gfCNCPoint5[15643] = {X -1.0364, Y 9.9250, Z -7.1667, A 0.000, B 0.000, C 0.000 }
gfCNCPoint5[15644] = {X -0.1703, Y 9.5539, Z -7.1667, A 0.000, B 0.000, C 0.000 }
gfCNCPoint5[15645] = {X 0.7570, Y 9.3871, Z -7.1667, A 0.000, B 0.000, C 0.000 }
gfCNCPoint5[15646] = {X 1.6981, Y 9.4333, Z -7.1667, A 0.000, B 0.000, C 0.000 }
gfCNCPoint5[15647] = {X 2.6047, Y 9.6901, Z -7.1667, A 0.000, B 0.000, C 0.000 }
gfCNCPoint5[15648] = {X 3.5530, Y 9.2659, Z -7.1667, A 0.000, B 0.000, C 0.000 }
gfCNCPoint5[15649] = {X 5.6159, Y 8.4887, Z -7.1667, A 0.000, B 0.000, C 0.000 }
gfCNCPoint5[15650] = {X 7.7422, Y 7.9071, Z -7.1667, A 0.000, B 0.000, C 0.000 }
gfCNCPoint5[15651] = {X 9.9135, Y 7.5260, Z -7.1667, A 0.000, B 0.000, C 0.000 }
gfCNCPoint5[15652] = {X 12.1108, Y 7.3488, Z -7.1667, A 0.000, B 0.000, C 0.000 }
gfCNCPoint5[15653] = {X 14.3150, Y 7.3770, Z -7.1667, A 0.000, B 0.000, C 0.000 }
gfCNCPoint5[15654] = {X 16.5070, Y 7.6105, Z -7.1667, A 0.000, B 0.000, C 0.000 }
gfCNCPoint5[15655] = {X 18.2265, Y 7.9626, Z -7.1667, A 0.000, B 0.000, C 0.000 }
gfCNCPoint5[15656] = {X 19.9014, Y 8.4872, Z -7.1667, A 0.000, B 0.000, C 0.000 }
gfCNCPoint5[15657] = {X 21.5145, Y 9.1790, Z -7.1667, A 0.000, B 0.000, C 0.000 }
gfCNCPoint5[15658] = {X 23.0491, Y 10.0308, Z -7.1667, A 0.000, B 0.000, C 0.000 }
gfCNCPoint5[15659] = {X 24.4894, Y 11.0338, Z -7.1667, A 0.000, B 0.000, C 0.000 }
gfCNCPoint5[15660] = {X 25.5613, Y 11.9712, Z -7.1667, A 0.000, B 0.000, C 0.000 }
gfCNCPoint5[15661] = {X 26.5229, Y 13.0215, Z -7.1667, A 0.000, B 0.000, C 0.000 }
gfCNCPoint5[15662] = {X 27.3624, Y 14.1717, Z -7.1667, A 0.000, B 0.000, C 0.000 }
gfCNCPoint5[15663] = {X 28.0693, Y 15.4079, Z -7.1667, A 0.000, B 0.000, C 0.000 }
gfCNCPoint5[15664] = {X 28.6351, Y 16.7147, Z -7.1667, A 0.000, B 0.000, C 0.000 }
gfCNCPoint5[15665] = {X 29.1044, Y 18.3529, Z -7.1667, A 0.000, B 0.000, C 0.000 }
gfCNCPoint5[15666] = {X 29.3828, Y 20.0341, Z -7.1667, A 0.000, B 0.000, C 0.000 }
gfCNCPoint5[15667] = {X 29.4668, Y 21.7361, Z -7.1667, A 0.000, B 0.000, C 0.000 }
gfCNCPoint5[15668] = {X 29.3551, Y 23.4365, Z -7.1667, A 0.000, B 0.000, C 0.000 }
gfCNCPoint5[15669] = {X 29.0493, Y 25.1129, Z -7.1667, A 0.000, B 0.000, C 0.000 }
gfCNCPoint5[15670] = {X 28.6229, Y 26.5132, Z -7.1667, A 0.000, B 0.000, C 0.000 }
gfCNCPoint5[15671] = {X 28.0227, Y 27.8482, Z -7.1667, A 0.000, B 0.000, C 0.000 }
gfCNCPoint5[15672] = {X 27.2582, Y 29.0964, Z -7.1667, A 0.000, B 0.000, C 0.000 }
gfCNCPoint5[15673] = {X 26.3417, Y 30.2377, Z -7.1667, A 0.000, B 0.000, C 0.000 }
gfCNCPoint5[15674] = {X 25.2881, Y 31.2538, Z -7.1667, A 0.000, B 0.000, C 0.000 }
gfCNCPoint5[15675] = {X 25.1139, Y 31.3987, Z -7.1667, A 0.000, B 0.000, C 0.000 }
gfCNCPoint5[15676] = {X 24.9369, Y 31.5402, Z -7.1667, A 0.000, B 0.000, C 0.000 }
gfCNCPoint5[15677] = {X 25.8030, Y 31.8442, Z -7.1667, A 0.000, B 0.000, C 0.000 }
gfCNCPoint5[15678] = {X 26.5813, Y 32.3308, Z -7.1667, A 0.000, B 0.000, C 0.000 }
gfCNCPoint5[15679] = {X 27.2339, Y 32.9762, Z -7.1667, A 0.000, B 0.000, C 0.000 }
gfCNCPoint5[15680] = {X 27.7292, Y 33.7491, Z -7.1667, A 0.000, B 0.000, C 0.000 }
gfCNCPoint5[15681] = {X 30.7660, Y 40.0227, Z -7.1667, A 0.000, B 0.000, C 0.000 }
gfCNCPoint5[15682] = {X 31.0747, Y 40.8982, Z -7.1667, A 0.000, B 0.000, C 0.000 }
gfCNCPoint5[15683] = {X 31.1815, Y 41.8203, Z -7.1667, A 0.000, B 0.000, C 0.000 }
gfCNCPoint5[15684] = {X 31.0813, Y 42.7431, Z -7.1667, A 0.000, B 0.000, C 0.000 }
gfCNCPoint5[15685] = {X 30.7789, Y 43.6208, Z -7.1667, A 0.000, B 0.000, C 0.000 }
gfCNCPoint5[15686] = {X 30.2893, Y 44.4095, Z -7.1667, A 0.000, B 0.000, C 0.000 }
gfCNCPoint5[15687] = {X 29.6371, Y 45.0700, Z -7.1667, A 0.000, B 0.000, C 0.000 }
gfCNCPoint5[15688] = {X 29.1011, Y 45.5034, Z -7.1667, A 0.000, B 0.000, C 0.000 }
gfCNCPoint5[15689] = {X 28.4112, Y 45.9565, Z -7.1667, A 0.000, B 0.000, C 0.000 }
gfCNCPoint5[15690] = {X 27.6455, Y 46.2648, Z -7.1667, A 0.000, B 0.000, C 0.000 }
gfCNCPoint5[15691] = {X 26.8342, Y 46.4162, Z -7.1667, A 0.000, B 0.000, C 0.000 }
gfCNCPoint5[15692] = {X 26.0089, Y 46.4050, Z -7.1667, A 0.000, B 0.000, C 0.000 }
gfCNCPoint5[15693] = {X 25.2019, Y 46.2314, Z -7.1667, A 0.000, B 0.000, C 0.000 }
gfCNCPoint5[15694] = {X 23.3925, Y 47.1909, Z -7.1667, A 0.000, B 0.000, C 0.000 }
gfCNCPoint5[15695] = {X 21.5199, Y 48.0206, Z -7.1667, A 0.000, B 0.000, C 0.000 }
gfCNCPoint5[15696] = {X 19.5936, Y 48.7163, Z -7.1667, A 0.000, B 0.000, C 0.000 }
gfCNCPoint5[15697] = {X 17.6674, Y 49.2600, Z -7.1667, A 0.000, B 0.000, C 0.000 }
gfCNCPoint5[15698] = {X 15.7006, Y 49.6311, Z -7.1667, A 0.000, B 0.000, C 0.000 }
gfCNCPoint5[15699] = {X 13.7087, Y 49.8267, Z -7.1667, A 0.000, B 0.000, C 0.000 }
gfCNCPoint5[15700] = {X 11.7074, Y 49.8453, Z -7.1667, A 0.000, B 0.000, C 0.000 }
gfCNCPoint5[15701] = {X 9.7122, Y 49.6868, Z -7.1667, A 0.000, B 0.000, C 0.000 }
gfCNCPoint5[15702] = {X 7.7389, Y 49.3523, Z -7.1667, A 0.000, B 0.000, C 0.000 }
gfCNCPoint5[15703] = {X 5.8554, Y 48.8363, Z -7.1667, A 0.000, B 0.000, C 0.000 }
gfCNCPoint5[15704] = {X 4.0458, Y 48.1022, Z -7.1667, A 0.000, B 0.000, C 0.000 }
gfCNCPoint5[15705] = {X 2.3352, Y 47.1601, Z -7.1667, A 0.000, B 0.000, C 0.000 }
gfCNCPoint5[15706] = {X 0.7475, Y 46.0231, Z -7.1667, A 0.000, B 0.000, C 0.000 }
gfCNCPoint5[15707] = {X -0.3710, Y 45.0177, Z -7.1667, A 0.000, B 0.000, C 0.000 }
gfCNCPoint5[15708] = {X -1.3644, Y 43.8885, Z -7.1667, A 0.000, B 0.000, C 0.000 }
gfCNCPoint5[15709] = {X -2.2192, Y 42.6512, Z -7.1667, A 0.000, B 0.000, C 0.000 }
gfCNCPoint5[15710] = {X -2.9237, Y 41.3225, Z -7.1667, A 0.000, B 0.000, C 0.000 }
gfCNCPoint5[15711] = {X -3.4683, Y 39.9206, Z -7.1667, A 0.000, B 0.000, C 0.000 }
gfCNCPoint5[15712] = {X -3.5888, Y 39.5251, Z -7.1667, A 0.000, B 0.000, C 0.000 }
gfCNCPoint5[15713] = {X -3.6967, Y 39.1259, Z -7.1667, A 0.000, B 0.000, C 0.000 }
gfCNCPoint5[15714] = {X -4.6774, Y 35.2480, Z -7.1667, A 0.000, B 0.000, C 0.000 }
gfCNCPoint5[15715] = {X -8.0069, Y 35.2272, Z -7.1667, A 0.000, B 0.000, C 0.000 }
gfCNCPoint5[15716] = {X -8.0069, Y 35.2272, Z -4.1667, A 0.000, B 0.000, C 0.000 }
gfCNCPoint5[15717] = {X -8.0069, Y 35.2272, Z 11.0000, A 0.000, B 0.000, C 0.000 }
gfCNCPoint5[15718] = {X -7.9995, Y 34.8056, Z 11.0000, A 0.000, B 0.000, C 0.000 }
gfCNCPoint5[15719] = {X -7.9995, Y 34.8056, Z -4.1667, A 0.000, B 0.000, C 0.000 }
gfCNCPoint5[15720] = {X -7.9995, Y 34.8056, Z -7.1667, A 0.000, B 0.000, C 0.000 }
gfCNCPoint5[15721] = {X -4.8517, Y 34.8970, Z -7.1667, A 0.000, B 0.000, C 0.000 }
gfCNCPoint5[15722] = {X -3.6967, Y 31.0674, Z -7.1667, A 0.000, B 0.000, C 0.000 }
gfCNCPoint5[15723] = {X -3.6591, Y 30.9448, Z -7.1667, A 0.000, B 0.000, C 0.000 }
gfCNCPoint5[15724] = {X -3.6205, Y 30.8225, Z -7.1667, A 0.000, B 0.000, C 0.000 }
gfCNCPoint5[15725] = {X -3.4458, Y 30.3101, Z -7.1667, A 0.000, B 0.000, C 0.000 }
gfCNCPoint5[15726] = {X -3.2526, Y 29.8045, Z -7.1667, A 0.000, B 0.000, C 0.000 }
gfCNCPoint5[15727] = {X -2.6179, Y 28.4651, Z -7.1667, A 0.000, B 0.000, C 0.000 }
gfCNCPoint5[15728] = {X -1.8063, Y 27.2249, Z -7.1667, A 0.000, B 0.000, C 0.000 }
gfCNCPoint5[15729] = {X -0.8329, Y 26.1072, Z -7.1667, A 0.000, B 0.000, C 0.000 }
gfCNCPoint5[15730] = {X 0.2840, Y 25.1328, Z -7.1667, A 0.000, B 0.000, C 0.000 }
gfCNCPoint5[15731] = {X 1.5235, Y 24.3201, Z -7.1667, A 0.000, B 0.000, C 0.000 }
gfCNCPoint5[15732] = {X 0.7354, Y 23.9293, Z -7.1667, A 0.000, B 0.000, C 0.000 }
gfCNCPoint5[15733] = {X 0.0428, Y 23.3868, Z -7.1667, A 0.000, B 0.000, C 0.000 }
gfCNCPoint5[15734] = {X -0.5255, Y 22.7154, Z -7.1667, A 0.000, B 0.000, C 0.000 }
gfCNCPoint5[15735] = {X -0.9460, Y 21.9427, Z -7.1667, A 0.000, B 0.000, C 0.000 }
gfCNCPoint5[15736] = {X -3.6217, Y 15.3839, Z -7.1667, A 0.000, B 0.000, C 0.000 }
gfCNCPoint5[15737] = {X -3.6606, Y 15.2745, Z -7.1667, A 0.000, B 0.000, C 0.000 }
gfCNCPoint5[15738] = {X -3.6967, Y 15.1642, Z -7.1667, A 0.000, B 0.000, C 0.000 }
gfCNCPoint5[15739] = {X -4.8865, Y 11.3452, Z -7.1667, A 0.000, B 0.000, C 0.000 }
gfCNCPoint5[15740] = {X -7.6967, Y 11.3452, Z -7.1667, A 0.000, B 0.000, C 0.000 }
gfCNCPoint5[15741] = {X -7.6967, Y 11.3452, Z -4.1667, A 0.000, B 0.000, C 0.000 }
gfCNCPoint5[15742] = {X -7.6967, Y 11.3452, Z 11.0000, A 0.000, B 0.000, C 0.000 }
gfCNCPoint5[15743] = {X -8.0065, Y 35.1744, Z 11.0000, A 0.000, B 0.000, C 0.000 }
gfCNCPoint5[15744] = {X -8.0065, Y 35.1744, Z -4.1667, A 0.000, B 0.000, C 0.000 }
gfCNCPoint5[15745] = {X -8.0065, Y 35.1744, Z -7.1667, A 0.000, B 0.000, C 0.000 }
gfCNCPoint5[15746] = {X -4.7803, Y 35.2037, Z -7.1667, A 0.000, B 0.000, C 0.000 }
gfCNCPoint5[15747] = {X -3.6967, Y 31.3533, Z -7.1667, A 0.000, B 0.000, C 0.000 }
gfCNCPoint5[15748] = {X -3.6228, Y 31.0994, Z -7.1667, A 0.000, B 0.000, C 0.000 }
gfCNCPoint5[15749] = {X -3.5443, Y 30.8469, Z -7.1667, A 0.000, B 0.000, C 0.000 }
gfCNCPoint5[15750] = {X -3.3705, Y 30.3371, Z -7.1667, A 0.000, B 0.000, C 0.000 }
gfCNCPoint5[15751] = {X -3.1782, Y 29.8341, Z -7.1667, A 0.000, B 0.000, C 0.000 }
gfCNCPoint5[15752] = {X -2.5643, Y 28.5332, Z -7.1667, A 0.000, B 0.000, C 0.000 }
gfCNCPoint5[15753] = {X -1.7821, Y 27.3259, Z -7.1667, A 0.000, B 0.000, C 0.000 }
gfCNCPoint5[15754] = {X -0.8458, Y 26.2339, Z -7.1667, A 0.000, B 0.000, C 0.000 }
gfCNCPoint5[15755] = {X 0.2280, Y 25.2767, Z -7.1667, A 0.000, B 0.000, C 0.000 }
gfCNCPoint5[15756] = {X 1.4199, Y 24.4715, Z -7.1667, A 0.000, B 0.000, C 0.000 }
gfCNCPoint5[15757] = {X 1.5687, Y 24.3865, Z -7.1667, A 0.000, B 0.000, C 0.000 }
gfCNCPoint5[15758] = {X 1.7187, Y 24.3039, Z -7.1667, A 0.000, B 0.000, C 0.000 }
gfCNCPoint5[15759] = {X 0.8916, Y 23.9307, Z -7.1667, A 0.000, B 0.000, C 0.000 }
gfCNCPoint5[15760] = {X 0.1628, Y 23.3900, Z -7.1667, A 0.000, B 0.000, C 0.000 }
gfCNCPoint5[15761] = {X -0.4342, Y 22.7066, Z -7.1667, A 0.000, B 0.000, C 0.000 }
gfCNCPoint5[15762] = {X -0.8722, Y 21.9118, Z -7.1667, A 0.000, B 0.000, C 0.000 }
gfCNCPoint5[15763] = {X -3.5467, Y 15.3560, Z -7.1667, A 0.000, B 0.000, C 0.000 }
gfCNCPoint5[15764] = {X -3.6292, Y 15.1114, Z -7.1667, A 0.000, B 0.000, C 0.000 }
gfCNCPoint5[15765] = {X -3.6967, Y 14.8622, Z -7.1667, A 0.000, B 0.000, C 0.000 }
gfCNCPoint5[15766] = {X -4.6241, Y 10.9713, Z -7.1667, A 0.000, B 0.000, C 0.000 }
gfCNCPoint5[15767] = {X -7.6967, Y 10.9713, Z -7.1667, A 0.000, B 0.000, C 0.000 }
gfCNCPoint5[15768] = {X -7.6967, Y 10.9713, Z -4.1667, A 0.000, B 0.000, C 0.000 }
gfCNCPoint5[15769] = {X -7.6967, Y 10.9713, Z 11.0000, A 0.000, B 0.000, C 0.000 }
gfCNCPoint5[15770] = {X -8.0058, Y 35.5721, Z 11.0000, A 0.000, B 0.000, C 0.000 }
gfCNCPoint5[15771] = {X -8.0058, Y 35.5721, Z -4.1667, A 0.000, B 0.000, C 0.000 }
gfCNCPoint5[15772] = {X -8.0058, Y 35.5721, Z -7.1667, A 0.000, B 0.000, C 0.000 }
gfCNCPoint5[15773] = {X -4.7025, Y 35.5310, Z -7.1667, A 0.000, B 0.000, C 0.000 }
gfCNCPoint5[15774] = {X -3.6967, Y 31.6595, Z -7.1667, A 0.000, B 0.000, C 0.000 }
gfCNCPoint5[15775] = {X -3.5879, Y 31.2638, Z -7.1667, A 0.000, B 0.000, C 0.000 }
gfCNCPoint5[15776] = {X -3.4681, Y 30.8713, Z -7.1667, A 0.000, B 0.000, C 0.000 }
gfCNCPoint5[15777] = {X -3.2952, Y 30.3642, Z -7.1667, A 0.000, B 0.000, C 0.000 }
gfCNCPoint5[15778] = {X -3.1039, Y 29.8636, Z -7.1667, A 0.000, B 0.000, C 0.000 }
gfCNCPoint5[15779] = {X -2.4945, Y 28.5724, Z -7.1667, A 0.000, B 0.000, C 0.000 }
gfCNCPoint5[15780] = {X -1.7182, Y 27.3740, Z -7.1667, A 0.000, B 0.000, C 0.000 }
gfCNCPoint5[15781] = {X -0.7888, Y 26.2901, Z -7.1667, A 0.000, B 0.000, C 0.000 }
gfCNCPoint5[15782] = {X 0.2770, Y 25.3399, Z -7.1667, A 0.000, B 0.000, C 0.000 }
gfCNCPoint5[15783] = {X 1.4602, Y 24.5406, Z -7.1667, A 0.000, B 0.000, C 0.000 }
gfCNCPoint5[15784] = {X 1.6926, Y 24.4092, Z -7.1667, A 0.000, B 0.000, C 0.000 }
gfCNCPoint5[15785] = {X 1.9282, Y 24.2837, Z -7.1667, A 0.000, B 0.000, C 0.000 }
gfCNCPoint5[15786] = {X 1.0580, Y 23.9328, Z -7.1667, A 0.000, B 0.000, C 0.000 }
gfCNCPoint5[15787] = {X 0.2886, Y 23.3958, Z -7.1667, A 0.000, B 0.000, C 0.000 }
gfCNCPoint5[15788] = {X -0.3408, Y 22.7000, Z -7.1667, A 0.000, B 0.000, C 0.000 }
gfCNCPoint5[15789] = {X -0.7984, Y 21.8809, Z -7.1667, A 0.000, B 0.000, C 0.000 }
gfCNCPoint5[15790] = {X -3.4717, Y 15.3281, Z -7.1667, A 0.000, B 0.000, C 0.000 }
gfCNCPoint5[15791] = {X -3.6097, Y 14.8813, Z -7.1667, A 0.000, B 0.000, C 0.000 }
gfCNCPoint5[15792] = {X -3.6967, Y 14.4218, Z -7.1667, A 0.000, B 0.000, C 0.000 }
gfCNCPoint5[15793] = {X -4.2185, Y 10.4560, Z -7.1667, A 0.000, B 0.000, C 0.000 }
gfCNCPoint5[15794] = {X -7.6967, Y 10.4560, Z -7.1667, A 0.000, B 0.000, C 0.000 }
gfCNCPoint5[15795] = {X -7.6967, Y 10.4560, Z -4.1667, A 0.000, B 0.000, C 0.000 }
gfCNCPoint5[15796] = {X -7.6967, Y 10.4560, Z 11.0000, A 0.000, B 0.000, C 0.000 }
gfCNCPoint5[15797] = {X -7.9953, Y 36.0059, Z 11.0000, A 0.000, B 0.000, C 0.000 }
gfCNCPoint5[15798] = {X -7.9953, Y 36.0059, Z -4.1667, A 0.000, B 0.000, C 0.000 }
gfCNCPoint5[15799] = {X -7.9953, Y 36.0059, Z -7.1667, A 0.000, B 0.000, C 0.000 }
gfCNCPoint5[15800] = {X -4.6168, Y 35.8845, Z -7.1667, A 0.000, B 0.000, C 0.000 }
gfCNCPoint5[15801] = {X -3.6967, Y 31.9918, Z -7.1667, A 0.000, B 0.000, C 0.000 }
gfCNCPoint5[15802] = {X -3.5550, Y 31.4408, Z -7.1667, A 0.000, B 0.000, C 0.000 }
gfCNCPoint5[15803] = {X -3.3919, Y 30.8958, Z -7.1667, A 0.000, B 0.000, C 0.000 }
gfCNCPoint5[15804] = {X -3.2199, Y 30.3912, Z -7.1667, A 0.000, B 0.000, C 0.000 }
gfCNCPoint5[15805] = {X -3.0296, Y 29.8932, Z -7.1667, A 0.000, B 0.000, C 0.000 }
gfCNCPoint5[15806] = {X -2.4248, Y 28.6115, Z -7.1667, A 0.000, B 0.000, C 0.000 }
gfCNCPoint5[15807] = {X -1.6542, Y 27.4221, Z -7.1667, A 0.000, B 0.000, C 0.000 }
gfCNCPoint5[15808] = {X -0.7318, Y 26.3462, Z -7.1667, A 0.000, B 0.000, C 0.000 }
gfCNCPoint5[15809] = {X 0.3261, Y 25.4031, Z -7.1667, A 0.000, B 0.000, C 0.000 }
gfCNCPoint5[15810] = {X 1.5004, Y 24.6098, Z -7.1667, A 0.000, B 0.000, C 0.000 }
gfCNCPoint5[15811] = {X 1.8254, Y 24.4282, Z -7.1667, A 0.000, B 0.000, C 0.000 }
gfCNCPoint5[15812] = {X 2.1565, Y 24.2581, Z -7.1667, A 0.000, B 0.000, C 0.000 }
gfCNCPoint5[15813] = {X 1.2383, Y 23.9358, Z -7.1667, A 0.000, B 0.000, C 0.000 }
gfCNCPoint5[15814] = {X 0.4225, Y 23.4052, Z -7.1667, A 0.000, B 0.000, C 0.000 }
gfCNCPoint5[15815] = {X -0.2445, Y 22.6965, Z -7.1667, A 0.000, B 0.000, C 0.000 }
gfCNCPoint5[15816] = {X -0.7246, Y 21.8500, Z -7.1667, A 0.000, B 0.000, C 0.000 }
gfCNCPoint5[15817] = {X -3.3967, Y 15.3003, Z -7.1667, A 0.000, B 0.000, C 0.000 }
gfCNCPoint5[15818] = {X -3.6236, Y 14.3619, Z -7.1667, A 0.000, B 0.000, C 0.000 }
gfCNCPoint5[15819] = {X -3.6236, Y 13.3964, Z -7.1667, A 0.000, B 0.000, C 0.000 }
gfCNCPoint5[15820] = {X -3.3967, Y 12.4580, Z -7.1667, A 0.000, B 0.000, C 0.000 }
gfCNCPoint5[15821] = {X -2.9671, Y 11.6161, Z -7.1667, A 0.000, B 0.000, C 0.000 }
gfCNCPoint5[15822] = {X -2.3552, Y 10.8956, Z -7.1667, A 0.000, B 0.000, C 0.000 }
gfCNCPoint5[15823] = {X -1.5940, Y 10.3353, Z -7.1667, A 0.000, B 0.000, C 0.000 }
gfCNCPoint5[15824] = {X -0.9967, Y 9.9945, Z -7.1667, A 0.000, B 0.000, C 0.000 }
gfCNCPoint5[15825] = {X -0.1386, Y 9.6279, Z -7.1667, A 0.000, B 0.000, C 0.000 }
gfCNCPoint5[15826] = {X 0.7805, Y 9.4658, Z -7.1667, A 0.000, B 0.000, C 0.000 }
gfCNCPoint5[15827] = {X 1.7123, Y 9.5168, Z -7.1667, A 0.000, B 0.000, C 0.000 }
gfCNCPoint5[15828] = {X 2.6082, Y 9.7782, Z -7.1667, A 0.000, B 0.000, C 0.000 }
gfCNCPoint5[15829] = {X 3.5852, Y 9.3391, Z -7.1667, A 0.000, B 0.000, C 0.000 }
gfCNCPoint5[15830] = {X 5.6410, Y 8.5647, Z -7.1667, A 0.000, B 0.000, C 0.000 }
gfCNCPoint5[15831] = {X 7.7601, Y 7.9850, Z -7.1667, A 0.000, B 0.000, C 0.000 }
gfCNCPoint5[15832] = {X 9.9239, Y 7.6053, Z -7.1667, A 0.000, B 0.000, C 0.000 }
gfCNCPoint5[15833] = {X 12.1137, Y 7.4287, Z -7.1667, A 0.000, B 0.000, C 0.000 }
gfCNCPoint5[15834] = {X 14.3104, Y 7.4569, Z -7.1667, A 0.000, B 0.000, C 0.000 }
gfCNCPoint5[15835] = {X 16.4949, Y 7.6895, Z -7.1667, A 0.000, B 0.000, C 0.000 }
gfCNCPoint5[15836] = {X 18.2064, Y 8.0400, Z -7.1667, A 0.000, B 0.000, C 0.000 }
gfCNCPoint5[15837] = {X 19.8736, Y 8.5622, Z -7.1667, A 0.000, B 0.000, C 0.000 }
gfCNCPoint5[15838] = {X 21.4792, Y 9.2508, Z -7.1667, A 0.000, B 0.000, C 0.000 }
gfCNCPoint5[15839] = {X 23.0067, Y 10.0987, Z -7.1667, A 0.000, B 0.000, C 0.000 }
gfCNCPoint5[15840] = {X 24.4404, Y 11.0971, Z -7.1667, A 0.000, B 0.000, C 0.000 }
gfCNCPoint5[15841] = {X 25.5055, Y 12.0285, Z -7.1667, A 0.000, B 0.000, C 0.000 }
gfCNCPoint5[15842] = {X 26.4610, Y 13.0721, Z -7.1667, A 0.000, B 0.000, C 0.000 }
gfCNCPoint5[15843] = {X 27.2951, Y 14.2150, Z -7.1667, A 0.000, B 0.000, C 0.000 }
gfCNCPoint5[15844] = {X 27.9976, Y 15.4433, Z -7.1667, A 0.000, B 0.000, C 0.000 }
gfCNCPoint5[15845] = {X 28.5598, Y 16.7417, Z -7.1667, A 0.000, B 0.000, C 0.000 }
gfCNCPoint5[15846] = {X 29.0264, Y 18.3710, Z -7.1667, A 0.000, B 0.000, C 0.000 }
gfCNCPoint5[15847] = {X 29.3033, Y 20.0431, Z -7.1667, A 0.000, B 0.000, C 0.000 }
gfCNCPoint5[15848] = {X 29.3868, Y 21.7358, Z -7.1667, A 0.000, B 0.000, C 0.000 }
gfCNCPoint5[15849] = {X 29.2757, Y 23.4270, Z -7.1667, A 0.000, B 0.000, C 0.000 }
gfCNCPoint5[15850] = {X 28.9715, Y 25.0943, Z -7.1667, A 0.000, B 0.000, C 0.000 }
gfCNCPoint5[15851] = {X 28.5481, Y 26.4849, Z -7.1667, A 0.000, B 0.000, C 0.000 }
gfCNCPoint5[15852] = {X 27.9520, Y 27.8107, Z -7.1667, A 0.000, B 0.000, C 0.000 }
gfCNCPoint5[15853] = {X 27.1928, Y 29.0503, Z -7.1667, A 0.000, B 0.000, C 0.000 }
gfCNCPoint5[15854] = {X 26.2827, Y 30.1837, Z -7.1667, A 0.000, B 0.000, C 0.000 }
gfCNCPoint5[15855] = {X 25.2363, Y 31.1928, Z -7.1667, A 0.000, B 0.000, C 0.000 }
gfCNCPoint5[15856] = {X 24.9961, Y 31.3912, Z -7.1667, A 0.000, B 0.000, C 0.000 }
gfCNCPoint5[15857] = {X 24.7505, Y 31.5830, Z -7.1667, A 0.000, B 0.000, C 0.000 }
gfCNCPoint5[15858] = {X 25.6511, Y 31.8623, Z -7.1667, A 0.000, B 0.000, C 0.000 }
gfCNCPoint5[15859] = {X 26.4636, Y 32.3409, Z -7.1667, A 0.000, B 0.000, C 0.000 }
gfCNCPoint5[15860] = {X 27.1445, Y 32.9933, Z -7.1667, A 0.000, B 0.000, C 0.000 }
gfCNCPoint5[15861] = {X 27.6575, Y 33.7845, Z -7.1667, A 0.000, B 0.000, C 0.000 }
gfCNCPoint5[15862] = {X 30.6940, Y 40.0576, Z -7.1667, A 0.000, B 0.000, C 0.000 }
gfCNCPoint5[15863] = {X 30.9967, Y 40.9162, Z -7.1667, A 0.000, B 0.000, C 0.000 }
gfCNCPoint5[15864] = {X 31.1015, Y 41.8206, Z -7.1667, A 0.000, B 0.000, C 0.000 }
gfCNCPoint5[15865] = {X 31.0032, Y 42.7257, Z -7.1667, A 0.000, B 0.000, C 0.000 }
gfCNCPoint5[15866] = {X 30.7066, Y 43.5864, Z -7.1667, A 0.000, B 0.000, C 0.000 }
gfCNCPoint5[15867] = {X 30.2265, Y 44.3600, Z -7.1667, A 0.000, B 0.000, C 0.000 }
gfCNCPoint5[15868] = {X 29.5868, Y 45.0078, Z -7.1667, A 0.000, B 0.000, C 0.000 }
gfCNCPoint5[15869] = {X 29.0508, Y 45.4412, Z -7.1667, A 0.000, B 0.000, C 0.000 }
gfCNCPoint5[15870] = {X 28.3678, Y 45.8889, Z -7.1667, A 0.000, B 0.000, C 0.000 }
gfCNCPoint5[15871] = {X 27.6096, Y 46.1919, Z -7.1667, A 0.000, B 0.000, C 0.000 }
gfCNCPoint5[15872] = {X 26.8062, Y 46.3383, Z -7.1667, A 0.000, B 0.000, C 0.000 }
gfCNCPoint5[15873] = {X 25.9898, Y 46.3222, Z -7.1667, A 0.000, B 0.000, C 0.000 }
gfCNCPoint5[15874] = {X 25.1928, Y 46.1442, Z -7.1667, A 0.000, B 0.000, C 0.000 }
gfCNCPoint5[15875] = {X 23.3788, Y 47.1086, Z -7.1667, A 0.000, B 0.000, C 0.000 }
gfCNCPoint5[15876] = {X 21.5009, Y 47.9420, Z -7.1667, A 0.000, B 0.000, C 0.000 }
gfCNCPoint5[15877] = {X 19.5687, Y 48.6402, Z -7.1667, A 0.000, B 0.000, C 0.000 }
gfCNCPoint5[15878] = {X 17.6493, Y 49.1820, Z -7.1667, A 0.000, B 0.000, C 0.000 }
gfCNCPoint5[15879] = {X 15.6895, Y 49.5519, Z -7.1667, A 0.000, B 0.000, C 0.000 }
gfCNCPoint5[15880] = {X 13.7046, Y 49.7468, Z -7.1667, A 0.000, B 0.000, C 0.000 }
gfCNCPoint5[15881] = {X 11.7102, Y 49.7654, Z -7.1667, A 0.000, B 0.000, C 0.000 }
gfCNCPoint5[15882] = {X 9.7221, Y 49.6074, Z -7.1667, A 0.000, B 0.000, C 0.000 }
gfCNCPoint5[15883] = {X 7.7557, Y 49.2741, Z -7.1667, A 0.000, B 0.000, C 0.000 }
gfCNCPoint5[15884] = {X 5.8812, Y 48.7606, Z -7.1667, A 0.000, B 0.000, C 0.000 }
gfCNCPoint5[15885] = {X 4.0802, Y 48.0299, Z -7.1667, A 0.000, B 0.000, C 0.000 }
gfCNCPoint5[15886] = {X 2.3778, Y 47.0923, Z -7.1667, A 0.000, B 0.000, C 0.000 }
gfCNCPoint5[15887] = {X 0.7976, Y 45.9608, Z -7.1667, A 0.000, B 0.000, C 0.000 }
gfCNCPoint5[15888] = {X -0.3139, Y 44.9616, Z -7.1667, A 0.000, B 0.000, C 0.000 }
gfCNCPoint5[15889] = {X -1.3012, Y 43.8394, Z -7.1667, A 0.000, B 0.000, C 0.000 }
gfCNCPoint5[15890] = {X -2.1507, Y 42.6097, Z -7.1667, A 0.000, B 0.000, C 0.000 }
gfCNCPoint5[15891] = {X -2.8509, Y 41.2892, Z -7.1667, A 0.000, B 0.000, C 0.000 }
gfCNCPoint5[15892] = {X -3.3921, Y 39.8960, Z -7.1667, A 0.000, B 0.000, C 0.000 }
gfCNCPoint5[15893] = {X -3.5570, Y 39.3424, Z -7.1667, A 0.000, B 0.000, C 0.000 }
gfCNCPoint5[15894] = {X -3.6967, Y 38.7818, Z -7.1667, A 0.000, B 0.000, C 0.000 }
gfCNCPoint5[15895] = {X -4.5759, Y 34.8796, Z -7.1667, A 0.000, B 0.000, C 0.000 }
gfCNCPoint5[15896] = {X -7.9985, Y 34.7745, Z -7.1667, A 0.000, B 0.000, C 0.000 }
gfCNCPoint5[15897] = {X -7.9985, Y 34.7745, Z -4.1667, A 0.000, B 0.000, C 0.000 }
gfCNCPoint5[15898] = {X -7.9985, Y 34.7745, Z 11.0000, A 0.000, B 0.000, C 0.000 }
gfCNCPoint5[15899] = {X -7.9718, Y 36.4871, Z 11.0000, A 0.000, B 0.000, C 0.000 }
gfCNCPoint5[15900] = {X -7.9718, Y 36.4871, Z -4.1667, A 0.000, B 0.000, C 0.000 }
gfCNCPoint5[15901] = {X -7.9718, Y 36.4871, Z -7.1667, A 0.000, B 0.000, C 0.000 }
gfCNCPoint5[15902] = {X -4.5206, Y 36.2729, Z -7.1667, A 0.000, B 0.000, C 0.000 }
gfCNCPoint5[15903] = {X -3.6967, Y 32.3587, Z -7.1667, A 0.000, B 0.000, C 0.000 }
gfCNCPoint5[15904] = {X -3.5247, Y 31.6345, Z -7.1667, A 0.000, B 0.000, C 0.000 }
gfCNCPoint5[15905] = {X -3.3158, Y 30.9202, Z -7.1667, A 0.000, B 0.000, C 0.000 }
gfCNCPoint5[15906] = {X -3.1443, Y 30.4173, Z -7.1667, A 0.000, B 0.000, C 0.000 }
gfCNCPoint5[15907] = {X -2.9545, Y 29.9211, Z -7.1667, A 0.000, B 0.000, C 0.000 }
gfCNCPoint5[15908] = {X -2.3543, Y 28.6494, Z -7.1667, A 0.000, B 0.000, C 0.000 }
gfCNCPoint5[15909] = {X -1.5896, Y 27.4693, Z -7.1667, A 0.000, B 0.000, C 0.000 }
gfCNCPoint5[15910] = {X -0.6743, Y 26.4018, Z -7.1667, A 0.000, B 0.000, C 0.000 }
gfCNCPoint5[15911] = {X 0.3754, Y 25.4661, Z -7.1667, A 0.000, B 0.000, C 0.000 }
gfCNCPoint5[15912] = {X 1.5407, Y 24.6789, Z -7.1667, A 0.000, B 0.000, C 0.000 }
gfCNCPoint5[15913] = {X 1.9707, Y 24.4419, Z -7.1667, A 0.000, B 0.000, C 0.000 }
gfCNCPoint5[15914] = {X 2.4113, Y 24.2252, Z -7.1667, A 0.000, B 0.000, C 0.000 }
gfCNCPoint5[15915] = {X 1.6198, Y 24.0145, Z -7.1667, A 0.000, B 0.000, C 0.000 }
gfCNCPoint5[15916] = {X 0.8879, Y 23.6470, Z -7.1667, A 0.000, B 0.000, C 0.000 }
gfCNCPoint5[15917] = {X 0.2461, Y 23.1382, Z -7.1667, A 0.000, B 0.000, C 0.000 }
gfCNCPoint5[15918] = {X -0.2786, Y 22.5093, Z -7.1667, A 0.000, B 0.000, C 0.000 }
gfCNCPoint5[15919] = {X -0.6642, Y 21.7867, Z -7.1667, A 0.000, B 0.000, C 0.000 }
gfCNCPoint5[15920] = {X -3.2754, Y 15.3911, Z -7.1667, A 0.000, B 0.000, C 0.000 }
gfCNCPoint5[15921] = {X -3.2991, Y 15.3319, Z -7.1667, A 0.000, B 0.000, C 0.000 }
gfCNCPoint5[15922] = {X -3.3217, Y 15.2724, Z -7.1667, A 0.000, B 0.000, C 0.000 }
gfCNCPoint5[15923] = {X -3.5441, Y 14.3524, Z -7.1667, A 0.000, B 0.000, C 0.000 }
gfCNCPoint5[15924] = {X -3.5441, Y 13.4059, Z -7.1667, A 0.000, B 0.000, C 0.000 }
gfCNCPoint5[15925] = {X -3.3217, Y 12.4858, Z -7.1667, A 0.000, B 0.000, C 0.000 }
gfCNCPoint5[15926] = {X -2.9005, Y 11.6604, Z -7.1667, A 0.000, B 0.000, C 0.000 }
gfCNCPoint5[15927] = {X -2.3006, Y 10.9541, Z -7.1667, A 0.000, B 0.000, C 0.000 }
gfCNCPoint5[15928] = {X -1.5544, Y 10.4048, Z -7.1667, A 0.000, B 0.000, C 0.000 }
gfCNCPoint5[15929] = {X -0.9063, Y 10.0355, Z -7.1667, A 0.000, B 0.000, C 0.000 }
gfCNCPoint5[15930] = {X -0.1051, Y 9.7014, Z -7.1667, A 0.000, B 0.000, C 0.000 }
gfCNCPoint5[15931] = {X 0.7492, Y 9.5480, Z -7.1667, A 0.000, B 0.000, C 0.000 }
gfCNCPoint5[15932] = {X 1.6165, Y 9.5825, Z -7.1667, A 0.000, B 0.000, C 0.000 }
gfCNCPoint5[15933] = {X 2.4560, Y 9.8032, Z -7.1667, A 0.000, B 0.000, C 0.000 }
gfCNCPoint5[15934] = {X 2.5433, Y 9.8378, Z -7.1667, A 0.000, B 0.000, C 0.000 }
gfCNCPoint5[15935] = {X 2.6297, Y 9.8745, Z -7.1667, A 0.000, B 0.000, C 0.000 }
gfCNCPoint5[15936] = {X 2.6555, Y 9.8427, Z -7.1667, A 0.000, B 0.000, C 0.000 }
gfCNCPoint5[15937] = {X 3.6169, Y 9.4126, Z -7.1667, A 0.000, B 0.000, C 0.000 }
gfCNCPoint5[15938] = {X 5.6658, Y 8.6407, Z -7.1667, A 0.000, B 0.000, C 0.000 }
gfCNCPoint5[15939] = {X 7.7777, Y 8.0631, Z -7.1667, A 0.000, B 0.000, C 0.000 }
gfCNCPoint5[15940] = {X 9.9343, Y 7.6846, Z -7.1667, A 0.000, B 0.000, C 0.000 }
gfCNCPoint5[15941] = {X 12.1167, Y 7.5087, Z -7.1667, A 0.000, B 0.000, C 0.000 }
gfCNCPoint5[15942] = {X 14.3060, Y 7.5368, Z -7.1667, A 0.000, B 0.000, C 0.000 }
gfCNCPoint5[15943] = {X 16.4832, Y 7.7687, Z -7.1667, A 0.000, B 0.000, C 0.000 }
gfCNCPoint5[15944] = {X 18.1867, Y 8.1175, Z -7.1667, A 0.000, B 0.000, C 0.000 }
gfCNCPoint5[15945] = {X 19.8460, Y 8.6373, Z -7.1667, A 0.000, B 0.000, C 0.000 }
gfCNCPoint5[15946] = {X 21.4441, Y 9.3227, Z -7.1667, A 0.000, B 0.000, C 0.000 }
gfCNCPoint5[15947] = {X 22.9644, Y 10.1666, Z -7.1667, A 0.000, B 0.000, C 0.000 }
gfCNCPoint5[15948] = {X 24.3914, Y 11.1603, Z -7.1667, A 0.000, B 0.000, C 0.000 }
gfCNCPoint5[15949] = {X 25.4497, Y 12.0858, Z -7.1667, A 0.000, B 0.000, C 0.000 }
gfCNCPoint5[15950] = {X 26.3990, Y 13.1227, Z -7.1667, A 0.000, B 0.000, C 0.000 }
gfCNCPoint5[15951] = {X 27.2278, Y 14.2583, Z -7.1667, A 0.000, B 0.000, C 0.000 }
gfCNCPoint5[15952] = {X 27.9258, Y 15.4786, Z -7.1667, A 0.000, B 0.000, C 0.000 }
gfCNCPoint5[15953] = {X 28.4845, Y 16.7687, Z -7.1667, A 0.000, B 0.000, C 0.000 }
gfCNCPoint5[15954] = {X 28.9486, Y 18.3893, Z -7.1667, A 0.000, B 0.000, C 0.000 }
gfCNCPoint5[15955] = {X 29.2239, Y 20.0524, Z -7.1667, A 0.000, B 0.000, C 0.000 }
gfCNCPoint5[15956] = {X 29.3068, Y 21.7361, Z -7.1667, A 0.000, B 0.000, C 0.000 }
gfCNCPoint5[15957] = {X 29.1961, Y 23.4182, Z -7.1667, A 0.000, B 0.000, C 0.000 }
gfCNCPoint5[15958] = {X 28.8934, Y 25.0766, Z -7.1667, A 0.000, B 0.000, C 0.000 }
gfCNCPoint5[15959] = {X 28.4730, Y 26.4573, Z -7.1667, A 0.000, B 0.000, C 0.000 }
gfCNCPoint5[15960] = {X 27.8811, Y 27.7737, Z -7.1667, A 0.000, B 0.000, C 0.000 }
gfCNCPoint5[15961] = {X 27.1272, Y 29.0045, Z -7.1667, A 0.000, B 0.000, C 0.000 }
gfCNCPoint5[15962] = {X 26.2235, Y 30.1299, Z -7.1667, A 0.000, B 0.000, C 0.000 }
gfCNCPoint5[15963] = {X 25.1846, Y 31.1318, Z -7.1667, A 0.000, B 0.000, C 0.000 }
gfCNCPoint5[15964] = {X 24.8725, Y 31.3873, Z -7.1667, A 0.000, B 0.000, C 0.000 }
gfCNCPoint5[15965] = {X 24.5516, Y 31.6316, Z -7.1667, A 0.000, B 0.000, C 0.000 }
gfCNCPoint5[15966] = {X 25.3139, Y 31.8152, Z -7.1667, A 0.000, B 0.000, C 0.000 }
gfCNCPoint5[15967] = {X 26.0258, Y 32.1441, Z -7.1667, A 0.000, B 0.000, C 0.000 }
gfCNCPoint5[15968] = {X 26.6598, Y 32.6056, Z -7.1667, A 0.000, B 0.000, C 0.000 }
gfCNCPoint5[15969] = {X 27.1916, Y 33.1818, Z -7.1667, A 0.000, B 0.000, C 0.000 }
gfCNCPoint5[15970] = {X 27.6008, Y 33.8508, Z -7.1667, A 0.000, B 0.000, C 0.000 }
gfCNCPoint5[15971] = {X 30.6220, Y 40.0925, Z -7.1667, A 0.000, B 0.000, C 0.000 }
gfCNCPoint5[15972] = {X 30.9188, Y 40.9342, Z -7.1667, A 0.000, B 0.000, C 0.000 }
gfCNCPoint5[15973] = {X 31.0215, Y 41.8209, Z -7.1667, A 0.000, B 0.000, C 0.000 }
gfCNCPoint5[15974] = {X 30.9251, Y 42.7082, Z -7.1667, A 0.000, B 0.000, C 0.000 }
gfCNCPoint5[15975] = {X 30.6343, Y 43.5521, Z -7.1667, A 0.000, B 0.000, C 0.000 }
gfCNCPoint5[15976] = {X 30.1637, Y 44.3105, Z -7.1667, A 0.000, B 0.000, C 0.000 }
gfCNCPoint5[15977] = {X 29.5365, Y 44.9456, Z -7.1667, A 0.000, B 0.000, C 0.000 }
gfCNCPoint5[15978] = {X 29.0005, Y 45.3790, Z -7.1667, A 0.000, B 0.000, C 0.000 }
gfCNCPoint5[15979] = {X 28.3245, Y 45.8212, Z -7.1667, A 0.000, B 0.000, C 0.000 }
gfCNCPoint5[15980] = {X 27.5737, Y 46.1190, Z -7.1667, A 0.000, B 0.000, C 0.000 }
gfCNCPoint5[15981] = {X 26.7784, Y 46.2602, Z -7.1667, A 0.000, B 0.000, C 0.000 }
gfCNCPoint5[15982] = {X 25.9709, Y 46.2392, Z -7.1667, A 0.000, B 0.000, C 0.000 }
gfCNCPoint5[15983] = {X 25.1840, Y 46.0569, Z -7.1667, A 0.000, B 0.000, C 0.000 }
gfCNCPoint5[15984] = {X 25.1083, Y 46.1006, Z -7.1667, A 0.000, B 0.000, C 0.000 }
gfCNCPoint5[15985] = {X 25.0325, Y 46.1441, Z -7.1667, A 0.000, B 0.000, C 0.000 }
gfCNCPoint5[15986] = {X 23.2604, Y 47.0771, Z -7.1667, A 0.000, B 0.000, C 0.000 }
gfCNCPoint5[15987] = {X 21.4280, Y 47.8850, Z -7.1667, A 0.000, B 0.000, C 0.000 }
gfCNCPoint5[15988] = {X 19.5440, Y 48.5641, Z -7.1667, A 0.000, B 0.000, C 0.000 }
gfCNCPoint5[15989] = {X 19.3883, Y 48.6154, Z -7.1667, A 0.000, B 0.000, C 0.000 }
gfCNCPoint5[15990] = {X 17.4982, Y 49.1352, Z -7.1667, A 0.000, B 0.000, C 0.000 }
gfCNCPoint5[15991] = {X 15.5700, Y 49.4881, Z -7.1667, A 0.000, B 0.000, C 0.000 }
gfCNCPoint5[15992] = {X 13.6183, Y 49.6714, Z -7.1667, A 0.000, B 0.000, C 0.000 }
gfCNCPoint5[15993] = {X 11.6581, Y 49.6835, Z -7.1667, A 0.000, B 0.000, C 0.000 }
gfCNCPoint5[15994] = {X 9.7042, Y 49.5246, Z -7.1667, A 0.000, B 0.000, C 0.000 }
gfCNCPoint5[15995] = {X 7.7718, Y 49.1957, Z -7.1667, A 0.000, B 0.000, C 0.000 }
gfCNCPoint5[15996] = {X 5.9062, Y 48.6846, Z -7.1667, A 0.000, B 0.000, C 0.000 }
gfCNCPoint5[15997] = {X 4.1138, Y 47.9573, Z -7.1667, A 0.000, B 0.000, C 0.000 }
gfCNCPoint5[15998] = {X 2.4195, Y 47.0240, Z -7.1667, A 0.000, B 0.000, C 0.000 }
gfCNCPoint5[15999] = {X 0.8469, Y 45.8977, Z -7.1667, A 0.000, B 0.000, C 0.000 }
gfCNCPoint5[16000] = {X -0.2575, Y 44.9048, Z -7.1667, A 0.000, B 0.000, C 0.000 }
gfCNCPoint5[16001] = {X -1.2384, Y 43.7898, Z -7.1667, A 0.000, B 0.000, C 0.000 }
gfCNCPoint5[16002] = {X -2.0825, Y 42.5679, Z -7.1667, A 0.000, B 0.000, C 0.000 }
gfCNCPoint5[16003] = {X -2.7782, Y 41.2558, Z -7.1667, A 0.000, B 0.000, C 0.000 }
gfCNCPoint5[16004] = {X -3.3160, Y 39.8715, Z -7.1667, A 0.000, B 0.000, C 0.000 }
gfCNCPoint5[16005] = {X -3.5286, Y 39.1374, Z -7.1667, A 0.000, B 0.000, C 0.000 }
gfCNCPoint5[16006] = {X -3.6967, Y 38.3919, Z -7.1667, A 0.000, B 0.000, C 0.000 }
gfCNCPoint5[16007] = {X -4.4586, Y 34.4652, Z -7.1667, A 0.000, B 0.000, C 0.000 }
gfCNCPoint5[16008] = {X -7.9755, Y 34.2587, Z -7.1667, A 0.000, B 0.000, C 0.000 }
gfCNCPoint5[16009] = {X -7.9755, Y 34.2587, Z -4.1667, A 0.000, B 0.000, C 0.000 }
gfCNCPoint5[16010] = {X -7.9755, Y 34.2587, Z 11.0000, A 0.000, B 0.000, C 0.000 }
gfCNCPoint5[16011] = {X 39.8243, Y 26.3831, Z 11.0000, A 0.000, B 0.000, C 0.000 }
gfCNCPoint5[16012] = {X 39.8243, Y 26.3831, Z -4.1667, A 0.000, B 0.000, C 0.000 }
gfCNCPoint5[16013] = {X 39.8243, Y 26.3831, Z -7.1667, A 0.000, B 0.000, C 0.000 }
gfCNCPoint5[16014] = {X 43.6477, Y 27.8073, Z -7.1667, A 0.000, B 0.000, C 0.000 }
gfCNCPoint5[16015] = {X 48.2901, Y 15.3446, Z -7.1667, A 0.000, B 0.000, C 0.000 }
gfCNCPoint5[16016] = {X 47.9079, Y 14.6186, Z -7.1667, A 0.000, B 0.000, C 0.000 }
gfCNCPoint5[16017] = {X 47.6697, Y 13.8334, Z -7.1667, A 0.000, B 0.000, C 0.000 }
gfCNCPoint5[16018] = {X 47.5844, Y 13.0173, Z -7.1667, A 0.000, B 0.000, C 0.000 }
gfCNCPoint5[16019] = {X 47.5842, Y 12.1868, Z -7.1667, A 0.000, B 0.000, C 0.000 }
gfCNCPoint5[16020] = {X 47.6925, Y 11.2255, Z -7.1667, A 0.000, B 0.000, C 0.000 }
gfCNCPoint5[16021] = {X 48.0120, Y 10.3125, Z -7.1667, A 0.000, B 0.000, C 0.000 }
gfCNCPoint5[16022] = {X 48.5267, Y 9.4933, Z -7.1667, A 0.000, B 0.000, C 0.000 }
gfCNCPoint5[16023] = {X 49.2107, Y 8.8093, Z -7.1667, A 0.000, B 0.000, C 0.000 }
gfCNCPoint5[16024] = {X 50.0298, Y 8.2946, Z -7.1667, A 0.000, B 0.000, C 0.000 }
gfCNCPoint5[16025] = {X 50.9429, Y 7.9751, Z -7.1667, A 0.000, B 0.000, C 0.000 }
gfCNCPoint5[16026] = {X 51.9042, Y 7.8668, Z -7.1667, A 0.000, B 0.000, C 0.000 }
gfCNCPoint5[16027] = {X 59.6221, Y 7.8668, Z -7.1667, A 0.000, B 0.000, C 0.000 }
gfCNCPoint5[16028] = {X 60.5834, Y 7.9751, Z -7.1667, A 0.000, B 0.000, C 0.000 }
gfCNCPoint5[16029] = {X 61.4965, Y 8.2946, Z -7.1667, A 0.000, B 0.000, C 0.000 }
gfCNCPoint5[16030] = {X 62.3156, Y 8.8093, Z -7.1667, A 0.000, B 0.000, C 0.000 }
gfCNCPoint5[16031] = {X 62.9996, Y 9.4933, Z -7.1667, A 0.000, B 0.000, C 0.000 }
gfCNCPoint5[16032] = {X 63.5143, Y 10.3124, Z -7.1667, A 0.000, B 0.000, C 0.000 }
gfCNCPoint5[16033] = {X 63.8338, Y 11.2255, Z -7.1667, A 0.000, B 0.000, C 0.000 }
gfCNCPoint5[16034] = {X 63.9421, Y 12.1868, Z -7.1667, A 0.000, B 0.000, C 0.000 }
gfCNCPoint5[16035] = {X 63.9421, Y 12.9782, Z -7.1667, A 0.000, B 0.000, C 0.000 }
gfCNCPoint5[16036] = {X 63.8584, Y 13.8244, Z -7.1667, A 0.000, B 0.000, C 0.000 }
gfCNCPoint5[16037] = {X 63.6106, Y 14.6378, Z -7.1667, A 0.000, B 0.000, C 0.000 }
gfCNCPoint5[16038] = {X 63.2082, Y 15.3869, Z -7.1667, A 0.000, B 0.000, C 0.000 }
gfCNCPoint5[16039] = {X 63.4268, Y 15.9633, Z -7.1667, A 0.000, B 0.000, C 0.000 }
gfCNCPoint5[16040] = {X 66.2401, Y 23.4301, Z -7.1667, A 0.000, B 0.000, C 0.000 }
gfCNCPoint5[16041] = {X 72.2107, Y 39.5004, Z -7.1667, A 0.000, B 0.000, C 0.000 }
gfCNCPoint5[16042] = {X 72.5162, Y 40.2688, Z -7.1667, A 0.000, B 0.000, C 0.000 }
gfCNCPoint5[16043] = {X 73.3602, Y 40.7707, Z -7.1667, A 0.000, B 0.000, C 0.000 }
gfCNCPoint5[16044] = {X 74.0691, Y 41.4503, Z -7.1667, A 0.000, B 0.000, C 0.000 }
gfCNCPoint5[16045] = {X 74.6062, Y 42.2724, Z -7.1667, A 0.000, B 0.000, C 0.000 }
gfCNCPoint5[16046] = {X 74.9437, Y 43.1946, Z -7.1667, A 0.000, B 0.000, C 0.000 }
gfCNCPoint5[16047] = {X 75.0643, Y 44.1692, Z -7.1667, A 0.000, B 0.000, C 0.000 }
gfCNCPoint5[16048] = {X 75.0645, Y 45.0000, Z -7.1667, A 0.000, B 0.000, C 0.000 }
gfCNCPoint5[16049] = {X 74.9561, Y 45.9613, Z -7.1667, A 0.000, B 0.000, C 0.000 }
gfCNCPoint5[16050] = {X 74.6366, Y 46.8744, Z -7.1667, A 0.000, B 0.000, C 0.000 }
gfCNCPoint5[16051] = {X 74.1220, Y 47.6935, Z -7.1667, A 0.000, B 0.000, C 0.000 }
gfCNCPoint5[16052] = {X 73.4379, Y 48.3775, Z -7.1667, A 0.000, B 0.000, C 0.000 }
gfCNCPoint5[16053] = {X 72.6188, Y 48.8922, Z -7.1667, A 0.000, B 0.000, C 0.000 }
gfCNCPoint5[16054] = {X 71.7057, Y 49.2117, Z -7.1667, A 0.000, B 0.000, C 0.000 }
gfCNCPoint5[16055] = {X 70.7445, Y 49.3200, Z -7.1667, A 0.000, B 0.000, C 0.000 }
gfCNCPoint5[16056] = {X 64.1851, Y 49.3200, Z -7.1667, A 0.000, B 0.000, C 0.000 }
gfCNCPoint5[16057] = {X 63.2238, Y 49.2117, Z -7.1667, A 0.000, B 0.000, C 0.000 }
gfCNCPoint5[16058] = {X 62.3108, Y 48.8922, Z -7.1667, A 0.000, B 0.000, C 0.000 }
gfCNCPoint5[16059] = {X 61.4917, Y 48.3775, Z -7.1667, A 0.000, B 0.000, C 0.000 }
gfCNCPoint5[16060] = {X 60.8076, Y 47.6935, Z -7.1667, A 0.000, B 0.000, C 0.000 }
gfCNCPoint5[16061] = {X 60.2930, Y 46.8744, Z -7.1667, A 0.000, B 0.000, C 0.000 }
gfCNCPoint5[16062] = {X 59.9734, Y 45.9613, Z -7.1667, A 0.000, B 0.000, C 0.000 }
gfCNCPoint5[16063] = {X 59.8651, Y 45.0000, Z -7.1667, A 0.000, B 0.000, C 0.000 }
gfCNCPoint5[16064] = {X 59.8651, Y 44.2085, Z -7.1667, A 0.000, B 0.000, C 0.000 }
gfCNCPoint5[16065] = {X 59.9516, Y 43.3503, Z -7.1667, A 0.000, B 0.000, C 0.000 }
gfCNCPoint5[16066] = {X 60.2069, Y 42.5263, Z -7.1667, A 0.000, B 0.000, C 0.000 }
gfCNCPoint5[16067] = {X 60.6208, Y 41.7695, Z -7.1667, A 0.000, B 0.000, C 0.000 }
gfCNCPoint5[16068] = {X 60.0065, Y 40.0892, Z -7.1667, A 0.000, B 0.000, C 0.000 }
gfCNCPoint5[16069] = {X 52.0782, Y 40.0892, Z -7.1667, A 0.000, B 0.000, C 0.000 }
gfCNCPoint5[16070] = {X 51.3351, Y 42.0858, Z -7.1667, A 0.000, B 0.000, C 0.000 }
gfCNCPoint5[16071] = {X 51.3381, Y 42.0907, Z -7.1667, A 0.000, B 0.000, C 0.000 }
gfCNCPoint5[16072] = {X 51.6392, Y 42.7500, Z -7.1667, A 0.000, B 0.000, C 0.000 }
gfCNCPoint5[16073] = {X 51.8258, Y 43.4503, Z -7.1667, A 0.000, B 0.000, C 0.000 }
gfCNCPoint5[16074] = {X 51.8928, Y 44.1720, Z -7.1667, A 0.000, B 0.000, C 0.000 }
gfCNCPoint5[16075] = {X 51.8929, Y 45.0000, Z -7.1667, A 0.000, B 0.000, C 0.000 }
gfCNCPoint5[16076] = {X 51.7846, Y 45.9613, Z -7.1667, A 0.000, B 0.000, C 0.000 }
gfCNCPoint5[16077] = {X 51.4651, Y 46.8744, Z -7.1667, A 0.000, B 0.000, C 0.000 }
gfCNCPoint5[16078] = {X 50.9504, Y 47.6935, Z -7.1667, A 0.000, B 0.000, C 0.000 }
gfCNCPoint5[16079] = {X 50.2664, Y 48.3775, Z -7.1667, A 0.000, B 0.000, C 0.000 }
gfCNCPoint5[16080] = {X 49.4473, Y 48.8922, Z -7.1667, A 0.000, B 0.000, C 0.000 }
gfCNCPoint5[16081] = {X 48.5342, Y 49.2117, Z -7.1667, A 0.000, B 0.000, C 0.000 }
gfCNCPoint5[16082] = {X 47.5729, Y 49.3200, Z -7.1667, A 0.000, B 0.000, C 0.000 }
gfCNCPoint5[16083] = {X 40.6393, Y 49.3200, Z -7.1667, A 0.000, B 0.000, C 0.000 }
gfCNCPoint5[16084] = {X 39.6780, Y 49.2117, Z -7.1667, A 0.000, B 0.000, C 0.000 }
gfCNCPoint5[16085] = {X 38.7649, Y 48.8922, Z -7.1667, A 0.000, B 0.000, C 0.000 }
gfCNCPoint5[16086] = {X 37.9458, Y 48.3775, Z -7.1667, A 0.000, B 0.000, C 0.000 }
gfCNCPoint5[16087] = {X 37.2618, Y 47.6935, Z -7.1667, A 0.000, B 0.000, C 0.000 }
gfCNCPoint5[16088] = {X 36.7471, Y 46.8744, Z -7.1667, A 0.000, B 0.000, C 0.000 }
gfCNCPoint5[16089] = {X 36.4276, Y 45.9613, Z -7.1667, A 0.000, B 0.000, C 0.000 }
gfCNCPoint5[16090] = {X 36.3193, Y 45.0000, Z -7.1667, A 0.000, B 0.000, C 0.000 }
gfCNCPoint5[16091] = {X 36.3193, Y 44.2086, Z -7.1667, A 0.000, B 0.000, C 0.000 }
gfCNCPoint5[16092] = {X 36.4359, Y 43.2117, Z -7.1667, A 0.000, B 0.000, C 0.000 }
gfCNCPoint5[16093] = {X 36.7795, Y 42.2686, Z -7.1667, A 0.000, B 0.000, C 0.000 }
gfCNCPoint5[16094] = {X 37.3314, Y 41.4303, Z -7.1667, A 0.000, B 0.000, C 0.000 }
gfCNCPoint5[16095] = {X 38.0618, Y 40.7420, Z -7.1667, A 0.000, B 0.000, C 0.000 }
gfCNCPoint5[16096] = {X 38.9314, Y 40.2407, Z -7.1667, A 0.000, B 0.000, C 0.000 }
gfCNCPoint5[16097] = {X 39.5223, Y 38.8449, Z -7.1667, A 0.000, B 0.000, C 0.000 }
gfCNCPoint5[16098] = {X 40.0635, Y 37.4290, Z -7.1667, A 0.000, B 0.000, C 0.000 }
gfCNCPoint5[16099] = {X 43.6477, Y 27.8073, Z -7.1667, A 0.000, B 0.000, C 0.000 }
gfCNCPoint5[16100] = {X 39.8993, Y 26.4110, Z -7.1667, A 0.000, B 0.000, C 0.000 }
gfCNCPoint5[16101] = {X 43.7226, Y 27.8352, Z -7.1667, A 0.000, B 0.000, C 0.000 }
gfCNCPoint5[16102] = {X 48.3793, Y 15.3344, Z -7.1667, A 0.000, B 0.000, C 0.000 }
gfCNCPoint5[16103] = {X 47.9922, Y 14.6130, Z -7.1667, A 0.000, B 0.000, C 0.000 }
gfCNCPoint5[16104] = {X 47.7508, Y 13.8307, Z -7.1667, A 0.000, B 0.000, C 0.000 }
gfCNCPoint5[16105] = {X 47.6644, Y 13.0166, Z -7.1667, A 0.000, B 0.000, C 0.000 }
gfCNCPoint5[16106] = {X 47.6642, Y 12.1868, Z -7.1667, A 0.000, B 0.000, C 0.000 }
gfCNCPoint5[16107] = {X 47.7705, Y 11.2433, Z -7.1667, A 0.000, B 0.000, C 0.000 }
gfCNCPoint5[16108] = {X 48.0841, Y 10.3472, Z -7.1667, A 0.000, B 0.000, C 0.000 }
gfCNCPoint5[16109] = {X 48.5893, Y 9.5432, Z -7.1667, A 0.000, B 0.000, C 0.000 }
gfCNCPoint5[16110] = {X 49.2606, Y 8.8719, Z -7.1667, A 0.000, B 0.000, C 0.000 }
gfCNCPoint5[16111] = {X 50.0646, Y 8.3667, Z -7.1667, A 0.000, B 0.000, C 0.000 }
gfCNCPoint5[16112] = {X 50.9607, Y 8.0531, Z -7.1667, A 0.000, B 0.000, C 0.000 }
gfCNCPoint5[16113] = {X 51.9042, Y 7.9468, Z -7.1667, A 0.000, B 0.000, C 0.000 }
gfCNCPoint5[16114] = {X 59.6221, Y 7.9468, Z -7.1667, A 0.000, B 0.000, C 0.000 }
gfCNCPoint5[16115] = {X 60.5656, Y 8.0531, Z -7.1667, A 0.000, B 0.000, C 0.000 }
gfCNCPoint5[16116] = {X 61.4618, Y 8.3667, Z -7.1667, A 0.000, B 0.000, C 0.000 }
gfCNCPoint5[16117] = {X 62.2657, Y 8.8718, Z -7.1667, A 0.000, B 0.000, C 0.000 }
gfCNCPoint5[16118] = {X 62.9371, Y 9.5432, Z -7.1667, A 0.000, B 0.000, C 0.000 }
gfCNCPoint5[16119] = {X 63.4422, Y 10.3471, Z -7.1667, A 0.000, B 0.000, C 0.000 }
gfCNCPoint5[16120] = {X 63.7558, Y 11.2433, Z -7.1667, A 0.000, B 0.000, C 0.000 }
gfCNCPoint5[16121] = {X 63.8621, Y 12.1868, Z -7.1667, A 0.000, B 0.000, C 0.000 }
gfCNCPoint5[16122] = {X 63.8621, Y 12.9782, Z -7.1667, A 0.000, B 0.000, C 0.000 }
gfCNCPoint5[16123] = {X 63.7772, Y 13.8222, Z -7.1667, A 0.000, B 0.000, C 0.000 }
gfCNCPoint5[16124] = {X 63.5261, Y 14.6324, Z -7.1667, A 0.000, B 0.000, C 0.000 }
gfCNCPoint5[16125] = {X 63.1186, Y 15.3764, Z -7.1667, A 0.000, B 0.000, C 0.000 }
gfCNCPoint5[16126] = {X 63.3519, Y 15.9916, Z -7.1667, A 0.000, B 0.000, C 0.000 }
gfCNCPoint5[16127] = {X 66.1652, Y 23.4582, Z -7.1667, A 0.000, B 0.000, C 0.000 }
gfCNCPoint5[16128] = {X 72.1360, Y 39.5291, Z -7.1667, A 0.000, B 0.000, C 0.000 }
gfCNCPoint5[16129] = {X 72.4539, Y 40.3287, Z -7.1667, A 0.000, B 0.000, C 0.000 }
gfCNCPoint5[16130] = {X 73.2912, Y 40.8188, Z -7.1667, A 0.000, B 0.000, C 0.000 }
gfCNCPoint5[16131] = {X 73.9951, Y 41.4865, Z -7.1667, A 0.000, B 0.000, C 0.000 }
gfCNCPoint5[16132] = {X 74.5289, Y 42.2968, Z -7.1667, A 0.000, B 0.000, C 0.000 }
gfCNCPoint5[16133] = {X 74.8644, Y 43.2071, Z -7.1667, A 0.000, B 0.000, C 0.000 }
gfCNCPoint5[16134] = {X 74.9843, Y 44.1699, Z -7.1667, A 0.000, B 0.000, C 0.000 }
gfCNCPoint5[16135] = {X 74.9845, Y 45.0000, Z -7.1667, A 0.000, B 0.000, C 0.000 }
gfCNCPoint5[16136] = {X 74.8782, Y 45.9435, Z -7.1667, A 0.000, B 0.000, C 0.000 }
gfCNCPoint5[16137] = {X 74.5646, Y 46.8397, Z -7.1667, A 0.000, B 0.000, C 0.000 }
gfCNCPoint5[16138] = {X 74.0594, Y 47.6436, Z -7.1667, A 0.000, B 0.000, C 0.000 }
gfCNCPoint5[16139] = {X 73.3881, Y 48.3150, Z -7.1667, A 0.000, B 0.000, C 0.000 }
gfCNCPoint5[16140] = {X 72.5841, Y 48.8201, Z -7.1667, A 0.000, B 0.000, C 0.000 }
gfCNCPoint5[16141] = {X 71.6879, Y 49.1337, Z -7.1667, A 0.000, B 0.000, C 0.000 }
gfCNCPoint5[16142] = {X 70.7445, Y 49.2400, Z -7.1667, A 0.000, B 0.000, C 0.000 }
gfCNCPoint5[16143] = {X 64.1851, Y 49.2400, Z -7.1667, A 0.000, B 0.000, C 0.000 }
gfCNCPoint5[16144] = {X 63.2416, Y 49.1337, Z -7.1667, A 0.000, B 0.000, C 0.000 }
gfCNCPoint5[16145] = {X 62.3455, Y 48.8201, Z -7.1667, A 0.000, B 0.000, C 0.000 }
gfCNCPoint5[16146] = {X 61.5415, Y 48.3150, Z -7.1667, A 0.000, B 0.000, C 0.000 }
gfCNCPoint5[16147] = {X 60.8702, Y 47.6436, Z -7.1667, A 0.000, B 0.000, C 0.000 }
gfCNCPoint5[16148] = {X 60.3650, Y 46.8397, Z -7.1667, A 0.000, B 0.000, C 0.000 }
gfCNCPoint5[16149] = {X 60.0514, Y 45.9435, Z -7.1667, A 0.000, B 0.000, C 0.000 }
gfCNCPoint5[16150] = {X 59.9451, Y 45.0000, Z -7.1667, A 0.000, B 0.000, C 0.000 }
gfCNCPoint5[16151] = {X 59.9451, Y 44.2085, Z -7.1667, A 0.000, B 0.000, C 0.000 }
gfCNCPoint5[16152] = {X 60.0328, Y 43.3528, Z -7.1667, A 0.000, B 0.000, C 0.000 }
gfCNCPoint5[16153] = {X 60.2913, Y 42.5323, Z -7.1667, A 0.000, B 0.000, C 0.000 }
gfCNCPoint5[16154] = {X 60.7101, Y 41.7810, Z -7.1667, A 0.000, B 0.000, C 0.000 }
gfCNCPoint5[16155] = {X 60.0624, Y 40.0092, Z -7.1667, A 0.000, B 0.000, C 0.000 }
gfCNCPoint5[16156] = {X 52.0226, Y 40.0092, Z -7.1667, A 0.000, B 0.000, C 0.000 }
gfCNCPoint5[16157] = {X 51.2468, Y 42.0937, Z -7.1667, A 0.000, B 0.000, C 0.000 }
gfCNCPoint5[16158] = {X 51.2688, Y 42.1307, Z -7.1667, A 0.000, B 0.000, C 0.000 }
gfCNCPoint5[16159] = {X 51.5641, Y 42.7776, Z -7.1667, A 0.000, B 0.000, C 0.000 }
gfCNCPoint5[16160] = {X 51.7471, Y 43.4646, Z -7.1667, A 0.000, B 0.000, C 0.000 }
gfCNCPoint5[16161] = {X 51.8128, Y 44.1726, Z -7.1667, A 0.000, B 0.000, C 0.000 }
gfCNCPoint5[16162] = {X 51.8129, Y 45.0000, Z -7.1667, A 0.000, B 0.000, C 0.000 }
gfCNCPoint5[16163] = {X 51.7066, Y 45.9435, Z -7.1667, A 0.000, B 0.000, C 0.000 }
gfCNCPoint5[16164] = {X 51.3930, Y 46.8397, Z -7.1667, A 0.000, B 0.000, C 0.000 }
gfCNCPoint5[16165] = {X 50.8879, Y 47.6436, Z -7.1667, A 0.000, B 0.000, C 0.000 }
gfCNCPoint5[16166] = {X 50.2165, Y 48.3150, Z -7.1667, A 0.000, B 0.000, C 0.000 }
gfCNCPoint5[16167] = {X 49.4126, Y 48.8201, Z -7.1667, A 0.000, B 0.000, C 0.000 }
gfCNCPoint5[16168] = {X 48.5164, Y 49.1337, Z -7.1667, A 0.000, B 0.000, C 0.000 }
gfCNCPoint5[16169] = {X 47.5729, Y 49.2400, Z -7.1667, A 0.000, B 0.000, C 0.000 }
gfCNCPoint5[16170] = {X 40.6393, Y 49.2400, Z -7.1667, A 0.000, B 0.000, C 0.000 }
gfCNCPoint5[16171] = {X 39.6958, Y 49.1337, Z -7.1667, A 0.000, B 0.000, C 0.000 }
gfCNCPoint5[16172] = {X 38.7996, Y 48.8201, Z -7.1667, A 0.000, B 0.000, C 0.000 }
gfCNCPoint5[16173] = {X 37.9957, Y 48.3150, Z -7.1667, A 0.000, B 0.000, C 0.000 }
gfCNCPoint5[16174] = {X 37.3243, Y 47.6436, Z -7.1667, A 0.000, B 0.000, C 0.000 }
gfCNCPoint5[16175] = {X 36.8192, Y 46.8397, Z -7.1667, A 0.000, B 0.000, C 0.000 }
gfCNCPoint5[16176] = {X 36.5056, Y 45.9435, Z -7.1667, A 0.000, B 0.000, C 0.000 }
gfCNCPoint5[16177] = {X 36.3993, Y 45.0000, Z -7.1667, A 0.000, B 0.000, C 0.000 }
gfCNCPoint5[16178] = {X 36.3993, Y 44.2086, Z -7.1667, A 0.000, B 0.000, C 0.000 }
gfCNCPoint5[16179] = {X 36.5152, Y 43.2241, Z -7.1667, A 0.000, B 0.000, C 0.000 }
gfCNCPoint5[16180] = {X 36.8566, Y 42.2934, Z -7.1667, A 0.000, B 0.000, C 0.000 }
gfCNCPoint5[16181] = {X 37.4047, Y 41.4675, Z -7.1667, A 0.000, B 0.000, C 0.000 }
gfCNCPoint5[16182] = {X 38.1296, Y 40.7913, Z -7.1667, A 0.000, B 0.000, C 0.000 }
gfCNCPoint5[16183] = {X 38.9917, Y 40.3020, Z -7.1667, A 0.000, B 0.000, C 0.000 }
gfCNCPoint5[16184] = {X 39.5906, Y 38.8894, Z -7.1667, A 0.000, B 0.000, C 0.000 }
gfCNCPoint5[16185] = {X 40.1387, Y 37.4562, Z -7.1667, A 0.000, B 0.000, C 0.000 }
gfCNCPoint5[16186] = {X 43.7226, Y 27.8352, Z -7.1667, A 0.000, B 0.000, C 0.000 }
gfCNCPoint5[16187] = {X 39.9743, Y 26.4389, Z -7.1667, A 0.000, B 0.000, C 0.000 }
gfCNCPoint5[16188] = {X 43.7976, Y 27.8632, Z -7.1667, A 0.000, B 0.000, C 0.000 }
gfCNCPoint5[16189] = {X 48.4687, Y 15.3238, Z -7.1667, A 0.000, B 0.000, C 0.000 }
gfCNCPoint5[16190] = {X 48.0765, Y 14.6072, Z -7.1667, A 0.000, B 0.000, C 0.000 }
gfCNCPoint5[16191] = {X 47.8320, Y 13.8279, Z -7.1667, A 0.000, B 0.000, C 0.000 }
gfCNCPoint5[16192] = {X 47.7444, Y 13.0158, Z -7.1667, A 0.000, B 0.000, C 0.000 }
gfCNCPoint5[16193] = {X 47.7442, Y 12.1868, Z -7.1667, A 0.000, B 0.000, C 0.000 }
gfCNCPoint5[16194] = {X 47.8485, Y 11.2611, Z -7.1667, A 0.000, B 0.000, C 0.000 }
gfCNCPoint5[16195] = {X 48.1562, Y 10.3819, Z -7.1667, A 0.000, B 0.000, C 0.000 }
gfCNCPoint5[16196] = {X 48.6518, Y 9.5931, Z -7.1667, A 0.000, B 0.000, C 0.000 }
gfCNCPoint5[16197] = {X 49.3105, Y 8.9344, Z -7.1667, A 0.000, B 0.000, C 0.000 }
gfCNCPoint5[16198] = {X 50.0993, Y 8.4388, Z -7.1667, A 0.000, B 0.000, C 0.000 }
gfCNCPoint5[16199] = {X 50.9785, Y 8.1311, Z -7.1667, A 0.000, B 0.000, C 0.000 }
gfCNCPoint5[16200] = {X 51.9042, Y 8.0268, Z -7.1667, A 0.000, B 0.000, C 0.000 }
gfCNCPoint5[16201] = {X 59.6221, Y 8.0268, Z -7.1667, A 0.000, B 0.000, C 0.000 }
gfCNCPoint5[16202] = {X 60.5478, Y 8.1311, Z -7.1667, A 0.000, B 0.000, C 0.000 }
gfCNCPoint5[16203] = {X 61.4271, Y 8.4388, Z -7.1667, A 0.000, B 0.000, C 0.000 }
gfCNCPoint5[16204] = {X 62.2158, Y 8.9344, Z -7.1667, A 0.000, B 0.000, C 0.000 }
gfCNCPoint5[16205] = {X 62.8745, Y 9.5931, Z -7.1667, A 0.000, B 0.000, C 0.000 }
gfCNCPoint5[16206] = {X 63.3702, Y 10.3819, Z -7.1667, A 0.000, B 0.000, C 0.000 }
gfCNCPoint5[16207] = {X 63.6778, Y 11.2611, Z -7.1667, A 0.000, B 0.000, C 0.000 }
gfCNCPoint5[16208] = {X 63.7821, Y 12.1868, Z -7.1667, A 0.000, B 0.000, C 0.000 }
gfCNCPoint5[16209] = {X 63.7821, Y 12.9782, Z -7.1667, A 0.000, B 0.000, C 0.000 }
gfCNCPoint5[16210] = {X 63.6961, Y 13.8199, Z -7.1667, A 0.000, B 0.000, C 0.000 }
gfCNCPoint5[16211] = {X 63.4415, Y 14.6267, Z -7.1667, A 0.000, B 0.000, C 0.000 }
gfCNCPoint5[16212] = {X 63.0289, Y 15.3654, Z -7.1667, A 0.000, B 0.000, C 0.000 }
gfCNCPoint5[16213] = {X 63.2771, Y 16.0198, Z -7.1667, A 0.000, B 0.000, C 0.000 }
gfCNCPoint5[16214] = {X 66.0903, Y 23.4862, Z -7.1667, A 0.000, B 0.000, C 0.000 }
gfCNCPoint5[16215] = {X 72.0613, Y 39.5578, Z -7.1667, A 0.000, B 0.000, C 0.000 }
gfCNCPoint5[16216] = {X 72.3917, Y 40.3888, Z -7.1667, A 0.000, B 0.000, C 0.000 }
gfCNCPoint5[16217] = {X 73.2222, Y 40.8672, Z -7.1667, A 0.000, B 0.000, C 0.000 }
gfCNCPoint5[16218] = {X 73.9212, Y 41.5229, Z -7.1667, A 0.000, B 0.000, C 0.000 }
gfCNCPoint5[16219] = {X 74.4516, Y 42.3212, Z -7.1667, A 0.000, B 0.000, C 0.000 }
gfCNCPoint5[16220] = {X 74.7852, Y 43.2197, Z -7.1667, A 0.000, B 0.000, C 0.000 }
gfCNCPoint5[16221] = {X 74.9043, Y 44.1706, Z -7.1667, A 0.000, B 0.000, C 0.000 }
gfCNCPoint5[16222] = {X 74.9045, Y 45.0000, Z -7.1667, A 0.000, B 0.000, C 0.000 }
gfCNCPoint5[16223] = {X 74.8002, Y 45.9257, Z -7.1667, A 0.000, B 0.000, C 0.000 }
gfCNCPoint5[16224] = {X 74.4925, Y 46.8050, Z -7.1667, A 0.000, B 0.000, C 0.000 }
gfCNCPoint5[16225] = {X 73.9969, Y 47.5937, Z -7.1667, A 0.000, B 0.000, C 0.000 }
gfCNCPoint5[16226] = {X 73.3382, Y 48.2524, Z -7.1667, A 0.000, B 0.000, C 0.000 }
gfCNCPoint5[16227] = {X 72.5494, Y 48.7480, Z -7.1667, A 0.000, B 0.000, C 0.000 }
gfCNCPoint5[16228] = {X 71.6701, Y 49.0557, Z -7.1667, A 0.000, B 0.000, C 0.000 }
gfCNCPoint5[16229] = {X 70.7445, Y 49.1600, Z -7.1667, A 0.000, B 0.000, C 0.000 }
gfCNCPoint5[16230] = {X 64.1851, Y 49.1600, Z -7.1667, A 0.000, B 0.000, C 0.000 }
gfCNCPoint5[16231] = {X 63.2594, Y 49.0557, Z -7.1667, A 0.000, B 0.000, C 0.000 }
gfCNCPoint5[16232] = {X 62.3802, Y 48.7480, Z -7.1667, A 0.000, B 0.000, C 0.000 }
gfCNCPoint5[16233] = {X 61.5914, Y 48.2524, Z -7.1667, A 0.000, B 0.000, C 0.000 }
gfCNCPoint5[16234] = {X 60.9327, Y 47.5937, Z -7.1667, A 0.000, B 0.000, C 0.000 }
gfCNCPoint5[16235] = {X 60.4371, Y 46.8050, Z -7.1667, A 0.000, B 0.000, C 0.000 }
gfCNCPoint5[16236] = {X 60.1294, Y 45.9257, Z -7.1667, A 0.000, B 0.000, C 0.000 }
gfCNCPoint5[16237] = {X 60.0251, Y 45.0000, Z -7.1667, A 0.000, B 0.000, C 0.000 }
gfCNCPoint5[16238] = {X 60.0251, Y 44.2086, Z -7.1667, A 0.000, B 0.000, C 0.000 }
gfCNCPoint5[16239] = {X 60.1139, Y 43.3554, Z -7.1667, A 0.000, B 0.000, C 0.000 }
gfCNCPoint5[16240] = {X 60.3758, Y 42.5386, Z -7.1667, A 0.000, B 0.000, C 0.000 }
gfCNCPoint5[16241] = {X 60.7997, Y 41.7929, Z -7.1667, A 0.000, B 0.000, C 0.000 }
gfCNCPoint5[16242] = {X 60.1184, Y 39.9292, Z -7.1667, A 0.000, B 0.000, C 0.000 }
gfCNCPoint5[16243] = {X 51.9670, Y 39.9292, Z -7.1667, A 0.000, B 0.000, C 0.000 }
gfCNCPoint5[16244] = {X 51.1585, Y 42.1016, Z -7.1667, A 0.000, B 0.000, C 0.000 }
gfCNCPoint5[16245] = {X 51.1995, Y 42.1707, Z -7.1667, A 0.000, B 0.000, C 0.000 }
gfCNCPoint5[16246] = {X 51.4890, Y 42.8051, Z -7.1667, A 0.000, B 0.000, C 0.000 }
gfCNCPoint5[16247] = {X 51.6684, Y 43.4790, Z -7.1667, A 0.000, B 0.000, C 0.000 }
gfCNCPoint5[16248] = {X 51.7328, Y 44.1733, Z -7.1667, A 0.000, B 0.000, C 0.000 }
gfCNCPoint5[16249] = {X 51.7329, Y 45.0000, Z -7.1667, A 0.000, B 0.000, C 0.000 }
gfCNCPoint5[16250] = {X 51.6286, Y 45.9257, Z -7.1667, A 0.000, B 0.000, C 0.000 }
gfCNCPoint5[16251] = {X 51.3210, Y 46.8050, Z -7.1667, A 0.000, B 0.000, C 0.000 }
gfCNCPoint5[16252] = {X 50.8253, Y 47.5937, Z -7.1667, A 0.000, B 0.000, C 0.000 }
gfCNCPoint5[16253] = {X 50.1666, Y 48.2524, Z -7.1667, A 0.000, B 0.000, C 0.000 }
gfCNCPoint5[16254] = {X 49.3779, Y 48.7480, Z -7.1667, A 0.000, B 0.000, C 0.000 }
gfCNCPoint5[16255] = {X 48.4986, Y 49.0557, Z -7.1667, A 0.000, B 0.000, C 0.000 }
gfCNCPoint5[16256] = {X 47.5729, Y 49.1600, Z -7.1667, A 0.000, B 0.000, C 0.000 }
gfCNCPoint5[16257] = {X 40.6393, Y 49.1600, Z -7.1667, A 0.000, B 0.000, C 0.000 }
gfCNCPoint5[16258] = {X 39.7136, Y 49.0557, Z -7.1667, A 0.000, B 0.000, C 0.000 }
gfCNCPoint5[16259] = {X 38.8343, Y 48.7480, Z -7.1667, A 0.000, B 0.000, C 0.000 }
gfCNCPoint5[16260] = {X 38.0456, Y 48.2524, Z -7.1667, A 0.000, B 0.000, C 0.000 }
gfCNCPoint5[16261] = {X 37.3869, Y 47.5937, Z -7.1667, A 0.000, B 0.000, C 0.000 }
gfCNCPoint5[16262] = {X 36.8913, Y 46.8050, Z -7.1667, A 0.000, B 0.000, C 0.000 }
gfCNCPoint5[16263] = {X 36.5836, Y 45.9257, Z -7.1667, A 0.000, B 0.000, C 0.000 }
gfCNCPoint5[16264] = {X 36.4793, Y 45.0000, Z -7.1667, A 0.000, B 0.000, C 0.000 }
gfCNCPoint5[16265] = {X 36.4793, Y 44.2086, Z -7.1667, A 0.000, B 0.000, C 0.000 }
gfCNCPoint5[16266] = {X 36.5945, Y 43.2366, Z -7.1667, A 0.000, B 0.000, C 0.000 }
gfCNCPoint5[16267] = {X 36.9336, Y 42.3184, Z -7.1667, A 0.000, B 0.000, C 0.000 }
gfCNCPoint5[16268] = {X 37.4780, Y 41.5048, Z -7.1667, A 0.000, B 0.000, C 0.000 }
gfCNCPoint5[16269] = {X 38.1973, Y 40.8410, Z -7.1667, A 0.000, B 0.000, C 0.000 }
gfCNCPoint5[16270] = {X 39.0518, Y 40.3636, Z -7.1667, A 0.000, B 0.000, C 0.000 }
gfCNCPoint5[16271] = {X 39.6589, Y 38.9340, Z -7.1667, A 0.000, B 0.000, C 0.000 }
gfCNCPoint5[16272] = {X 40.2139, Y 37.4835, Z -7.1667, A 0.000, B 0.000, C 0.000 }
gfCNCPoint5[16273] = {X 43.7976, Y 27.8632, Z -7.1667, A 0.000, B 0.000, C 0.000 }
gfCNCPoint5[16274] = {X 40.0492, Y 26.4669, Z -7.1667, A 0.000, B 0.000, C 0.000 }
gfCNCPoint5[16275] = {X 43.8726, Y 27.8911, Z -7.1667, A 0.000, B 0.000, C 0.000 }
gfCNCPoint5[16276] = {X 48.5582, Y 15.3126, Z -7.1667, A 0.000, B 0.000, C 0.000 }
gfCNCPoint5[16277] = {X 48.1610, Y 14.6012, Z -7.1667, A 0.000, B 0.000, C 0.000 }
gfCNCPoint5[16278] = {X 47.9131, Y 13.8250, Z -7.1667, A 0.000, B 0.000, C 0.000 }
gfCNCPoint5[16279] = {X 47.8244, Y 13.0151, Z -7.1667, A 0.000, B 0.000, C 0.000 }
gfCNCPoint5[16280] = {X 47.8242, Y 12.1868, Z -7.1667, A 0.000, B 0.000, C 0.000 }
gfCNCPoint5[16281] = {X 47.9265, Y 11.2789, Z -7.1667, A 0.000, B 0.000, C 0.000 }
gfCNCPoint5[16282] = {X 48.2283, Y 10.4166, Z -7.1667, A 0.000, B 0.000, C 0.000 }
gfCNCPoint5[16283] = {X 48.7144, Y 9.6430, Z -7.1667, A 0.000, B 0.000, C 0.000 }
gfCNCPoint5[16284] = {X 49.3604, Y 8.9969, Z -7.1667, A 0.000, B 0.000, C 0.000 }
gfCNCPoint5[16285] = {X 50.1340, Y 8.5109, Z -7.1667, A 0.000, B 0.000, C 0.000 }
gfCNCPoint5[16286] = {X 50.9963, Y 8.2091, Z -7.1667, A 0.000, B 0.000, C 0.000 }
gfCNCPoint5[16287] = {X 51.9042, Y 8.1068, Z -7.1667, A 0.000, B 0.000, C 0.000 }
gfCNCPoint5[16288] = {X 59.6221, Y 8.1068, Z -7.1667, A 0.000, B 0.000, C 0.000 }
gfCNCPoint5[16289] = {X 60.5300, Y 8.2091, Z -7.1667, A 0.000, B 0.000, C 0.000 }
gfCNCPoint5[16290] = {X 61.3924, Y 8.5109, Z -7.1667, A 0.000, B 0.000, C 0.000 }
gfCNCPoint5[16291] = {X 62.1660, Y 8.9969, Z -7.1667, A 0.000, B 0.000, C 0.000 }
gfCNCPoint5[16292] = {X 62.8120, Y 9.6430, Z -7.1667, A 0.000, B 0.000, C 0.000 }
gfCNCPoint5[16293] = {X 63.2981, Y 10.4166, Z -7.1667, A 0.000, B 0.000, C 0.000 }
gfCNCPoint5[16294] = {X 63.5998, Y 11.2789, Z -7.1667, A 0.000, B 0.000, C 0.000 }
gfCNCPoint5[16295] = {X 63.7021, Y 12.1868, Z -7.1667, A 0.000, B 0.000, C 0.000 }
gfCNCPoint5[16296] = {X 63.7021, Y 12.9782, Z -7.1667, A 0.000, B 0.000, C 0.000 }
gfCNCPoint5[16297] = {X 63.6148, Y 13.8174, Z -7.1667, A 0.000, B 0.000, C 0.000 }
gfCNCPoint5[16298] = {X 63.3568, Y 14.6208, Z -7.1667, A 0.000, B 0.000, C 0.000 }
gfCNCPoint5[16299] = {X 62.9390, Y 15.3539, Z -7.1667, A 0.000, B 0.000, C 0.000 }
gfCNCPoint5[16300] = {X 63.2023, Y 16.0481, Z -7.1667, A 0.000, B 0.000, C 0.000 }
gfCNCPoint5[16301] = {X 66.0153, Y 23.5142, Z -7.1667, A 0.000, B 0.000, C 0.000 }
gfCNCPoint5[16302] = {X 71.9867, Y 39.5865, Z -7.1667, A 0.000, B 0.000, C 0.000 }
gfCNCPoint5[16303] = {X 72.3297, Y 40.4493, Z -7.1667, A 0.000, B 0.000, C 0.000 }
gfCNCPoint5[16304] = {X 73.1533, Y 40.9158, Z -7.1667, A 0.000, B 0.000, C 0.000 }
gfCNCPoint5[16305] = {X 73.8473, Y 41.5595, Z -7.1667, A 0.000, B 0.000, C 0.000 }
gfCNCPoint5[16306] = {X 74.3743, Y 42.3457, Z -7.1667, A 0.000, B 0.000, C 0.000 }
gfCNCPoint5[16307] = {X 74.7059, Y 43.2323, Z -7.1667, A 0.000, B 0.000, C 0.000 }
gfCNCPoint5[16308] = {X 74.8243, Y 44.1714, Z -7.1667, A 0.000, B 0.000, C 0.000 }
gfCNCPoint5[16309] = {X 74.8245, Y 45.0000, Z -7.1667, A 0.000, B 0.000, C 0.000 }
gfCNCPoint5[16310] = {X 74.7222, Y 45.9079, Z -7.1667, A 0.000, B 0.000, C 0.000 }
gfCNCPoint5[16311] = {X 74.4204, Y 46.7702, Z -7.1667, A 0.000, B 0.000, C 0.000 }
gfCNCPoint5[16312] = {X 73.9343, Y 47.5438, Z -7.1667, A 0.000, B 0.000, C 0.000 }
gfCNCPoint5[16313] = {X 73.2883, Y 48.1899, Z -7.1667, A 0.000, B 0.000, C 0.000 }
gfCNCPoint5[16314] = {X 72.5147, Y 48.6760, Z -7.1667, A 0.000, B 0.000, C 0.000 }
gfCNCPoint5[16315] = {X 71.6523, Y 48.9777, Z -7.1667, A 0.000, B 0.000, C 0.000 }
gfCNCPoint5[16316] = {X 70.7445, Y 49.0800, Z -7.1667, A 0.000, B 0.000, C 0.000 }
gfCNCPoint5[16317] = {X 64.1851, Y 49.0800, Z -7.1667, A 0.000, B 0.000, C 0.000 }
gfCNCPoint5[16318] = {X 63.2772, Y 48.9777, Z -7.1667, A 0.000, B 0.000, C 0.000 }
gfCNCPoint5[16319] = {X 62.4149, Y 48.6760, Z -7.1667, A 0.000, B 0.000, C 0.000 }
gfCNCPoint5[16320] = {X 61.6413, Y 48.1899, Z -7.1667, A 0.000, B 0.000, C 0.000 }
gfCNCPoint5[16321] = {X 60.9953, Y 47.5438, Z -7.1667, A 0.000, B 0.000, C 0.000 }
gfCNCPoint5[16322] = {X 60.5092, Y 46.7702, Z -7.1667, A 0.000, B 0.000, C 0.000 }
gfCNCPoint5[16323] = {X 60.2074, Y 45.9079, Z -7.1667, A 0.000, B 0.000, C 0.000 }
gfCNCPoint5[16324] = {X 60.1051, Y 45.0000, Z -7.1667, A 0.000, B 0.000, C 0.000 }
gfCNCPoint5[16325] = {X 60.1051, Y 44.2086, Z -7.1667, A 0.000, B 0.000, C 0.000 }
gfCNCPoint5[16326] = {X 60.1951, Y 43.3581, Z -7.1667, A 0.000, B 0.000, C 0.000 }
gfCNCPoint5[16327] = {X 60.4604, Y 42.5451, Z -7.1667, A 0.000, B 0.000, C 0.000 }
gfCNCPoint5[16328] = {X 60.8894, Y 41.8053, Z -7.1667, A 0.000, B 0.000, C 0.000 }
gfCNCPoint5[16329] = {X 60.1743, Y 39.8492, Z -7.1667, A 0.000, B 0.000, C 0.000 }
gfCNCPoint5[16330] = {X 51.9115, Y 39.8492, Z -7.1667, A 0.000, B 0.000, C 0.000 }
gfCNCPoint5[16331] = {X 51.0702, Y 42.1095, Z -7.1667, A 0.000, B 0.000, C 0.000 }
gfCNCPoint5[16332] = {X 51.1302, Y 42.2107, Z -7.1667, A 0.000, B 0.000, C 0.000 }
gfCNCPoint5[16333] = {X 51.4139, Y 42.8327, Z -7.1667, A 0.000, B 0.000, C 0.000 }
gfCNCPoint5[16334] = {X 51.5897, Y 43.4933, Z -7.1667, A 0.000, B 0.000, C 0.000 }
gfCNCPoint5[16335] = {X 51.6528, Y 44.1740, Z -7.1667, A 0.000, B 0.000, C 0.000 }
gfCNCPoint5[16336] = {X 51.6529, Y 45.0000, Z -7.1667, A 0.000, B 0.000, C 0.000 }
gfCNCPoint5[16337] = {X 51.5506, Y 45.9079, Z -7.1667, A 0.000, B 0.000, C 0.000 }
gfCNCPoint5[16338] = {X 51.2489, Y 46.7702, Z -7.1667, A 0.000, B 0.000, C 0.000 }
gfCNCPoint5[16339] = {X 50.7628, Y 47.5438, Z -7.1667, A 0.000, B 0.000, C 0.000 }
gfCNCPoint5[16340] = {X 50.1168, Y 48.1899, Z -7.1667, A 0.000, B 0.000, C 0.000 }
gfCNCPoint5[16341] = {X 49.3432, Y 48.6760, Z -7.1667, A 0.000, B 0.000, C 0.000 }
gfCNCPoint5[16342] = {X 48.4808, Y 48.9777, Z -7.1667, A 0.000, B 0.000, C 0.000 }
gfCNCPoint5[16343] = {X 47.5729, Y 49.0800, Z -7.1667, A 0.000, B 0.000, C 0.000 }
gfCNCPoint5[16344] = {X 40.6393, Y 49.0800, Z -7.1667, A 0.000, B 0.000, C 0.000 }
gfCNCPoint5[16345] = {X 39.7314, Y 48.9777, Z -7.1667, A 0.000, B 0.000, C 0.000 }
gfCNCPoint5[16346] = {X 38.8691, Y 48.6760, Z -7.1667, A 0.000, B 0.000, C 0.000 }
gfCNCPoint5[16347] = {X 38.0955, Y 48.1899, Z -7.1667, A 0.000, B 0.000, C 0.000 }
gfCNCPoint5[16348] = {X 37.4494, Y 47.5438, Z -7.1667, A 0.000, B 0.000, C 0.000 }
gfCNCPoint5[16349] = {X 36.9633, Y 46.7702, Z -7.1667, A 0.000, B 0.000, C 0.000 }
gfCNCPoint5[16350] = {X 36.6616, Y 45.9079, Z -7.1667, A 0.000, B 0.000, C 0.000 }
gfCNCPoint5[16351] = {X 36.5593, Y 45.0000, Z -7.1667, A 0.000, B 0.000, C 0.000 }
gfCNCPoint5[16352] = {X 36.5593, Y 44.2086, Z -7.1667, A 0.000, B 0.000, C 0.000 }
gfCNCPoint5[16353] = {X 36.6733, Y 43.2509, Z -7.1667, A 0.000, B 0.000, C 0.000 }
gfCNCPoint5[16354] = {X 37.0090, Y 42.3468, Z -7.1667, A 0.000, B 0.000, C 0.000 }
gfCNCPoint5[16355] = {X 37.5474, Y 41.5467, Z -7.1667, A 0.000, B 0.000, C 0.000 }
gfCNCPoint5[16356] = {X 38.2586, Y 40.8953, Z -7.1667, A 0.000, B 0.000, C 0.000 }
gfCNCPoint5[16357] = {X 39.1029, Y 40.4291, Z -7.1667, A 0.000, B 0.000, C 0.000 }
gfCNCPoint5[16358] = {X 39.1157, Y 40.4167, Z -7.1667, A 0.000, B 0.000, C 0.000 }
gfCNCPoint5[16359] = {X 39.1249, Y 40.3962, Z -7.1667, A 0.000, B 0.000, C 0.000 }
gfCNCPoint5[16360] = {X 39.7331, Y 38.9640, Z -7.1667, A 0.000, B 0.000, C 0.000 }
gfCNCPoint5[16361] = {X 40.2892, Y 37.5107, Z -7.1667, A 0.000, B 0.000, C 0.000 }
gfCNCPoint5[16362] = {X 43.8726, Y 27.8911, Z -7.1667, A 0.000, B 0.000, C 0.000 }
gfCNCPoint5[16363] = {X 40.1242, Y 26.4948, Z -7.1667, A 0.000, B 0.000, C 0.000 }
gfCNCPoint5[16364] = {X 43.9475, Y 27.9190, Z -7.1667, A 0.000, B 0.000, C 0.000 }
gfCNCPoint5[16365] = {X 48.6479, Y 15.3010, Z -7.1667, A 0.000, B 0.000, C 0.000 }
gfCNCPoint5[16366] = {X 48.2407, Y 14.5838, Z -7.1667, A 0.000, B 0.000, C 0.000 }
gfCNCPoint5[16367] = {X 47.9892, Y 13.7983, Z -7.1667, A 0.000, B 0.000, C 0.000 }
gfCNCPoint5[16368] = {X 47.9042, Y 12.9780, Z -7.1667, A 0.000, B 0.000, C 0.000 }
gfCNCPoint5[16369] = {X 47.9042, Y 12.1868, Z -7.1667, A 0.000, B 0.000, C 0.000 }
gfCNCPoint5[16370] = {X 48.0045, Y 11.2967, Z -7.1667, A 0.000, B 0.000, C 0.000 }
gfCNCPoint5[16371] = {X 48.3003, Y 10.4513, Z -7.1667, A 0.000, B 0.000, C 0.000 }
gfCNCPoint5[16372] = {X 48.7769, Y 9.6929, Z -7.1667, A 0.000, B 0.000, C 0.000 }
gfCNCPoint5[16373] = {X 49.4103, Y 9.0595, Z -7.1667, A 0.000, B 0.000, C 0.000 }
gfCNCPoint5[16374] = {X 50.1687, Y 8.5829, Z -7.1667, A 0.000, B 0.000, C 0.000 }
gfCNCPoint5[16375] = {X 51.0141, Y 8.2871, Z -7.1667, A 0.000, B 0.000, C 0.000 }
gfCNCPoint5[16376] = {X 51.9042, Y 8.1868, Z -7.1667, A 0.000, B 0.000, C 0.000 }
gfCNCPoint5[16377] = {X 59.6221, Y 8.1868, Z -7.1667, A 0.000, B 0.000, C 0.000 }
gfCNCPoint5[16378] = {X 60.5122, Y 8.2871, Z -7.1667, A 0.000, B 0.000, C 0.000 }
gfCNCPoint5[16379] = {X 61.3577, Y 8.5829, Z -7.1667, A 0.000, B 0.000, C 0.000 }
gfCNCPoint5[16380] = {X 62.1161, Y 9.0595, Z -7.1667, A 0.000, B 0.000, C 0.000 }
gfCNCPoint5[16381] = {X 62.7495, Y 9.6929, Z -7.1667, A 0.000, B 0.000, C 0.000 }
gfCNCPoint5[16382] = {X 63.2260, Y 10.4513, Z -7.1667, A 0.000, B 0.000, C 0.000 }
gfCNCPoint5[16383] = {X 63.5218, Y 11.2967, Z -7.1667, A 0.000, B 0.000, C 0.000 }
gfCNCPoint5[16384] = {X 63.6221, Y 12.1868, Z -7.1667, A 0.000, B 0.000, C 0.000 }
gfCNCPoint5[16385] = {X 63.6219, Y 13.0192, Z -7.1667, A 0.000, B 0.000, C 0.000 }
gfCNCPoint5[16386] = {X 63.5278, Y 13.8416, Z -7.1667, A 0.000, B 0.000, C 0.000 }
gfCNCPoint5[16387] = {X 63.2664, Y 14.6271, Z -7.1667, A 0.000, B 0.000, C 0.000 }
gfCNCPoint5[16388] = {X 62.8489, Y 15.3419, Z -7.1667, A 0.000, B 0.000, C 0.000 }
gfCNCPoint5[16389] = {X 63.1274, Y 16.0764, Z -7.1667, A 0.000, B 0.000, C 0.000 }
gfCNCPoint5[16390] = {X 65.9404, Y 23.5423, Z -7.1667, A 0.000, B 0.000, C 0.000 }
gfCNCPoint5[16391] = {X 71.9120, Y 39.6152, Z -7.1667, A 0.000, B 0.000, C 0.000 }
gfCNCPoint5[16392] = {X 72.2608, Y 40.4925, Z -7.1667, A 0.000, B 0.000, C 0.000 }
gfCNCPoint5[16393] = {X 72.2705, Y 40.5075, Z -7.1667, A 0.000, B 0.000, C 0.000 }
gfCNCPoint5[16394] = {X 72.2853, Y 40.5175, Z -7.1667, A 0.000, B 0.000, C 0.000 }
gfCNCPoint5[16395] = {X 72.3488, Y 40.5446, Z -7.1667, A 0.000, B 0.000, C 0.000 }
gfCNCPoint5[16396] = {X 72.4119, Y 40.5729, Z -7.1667, A 0.000, B 0.000, C 0.000 }
gfCNCPoint5[16397] = {X 73.1911, Y 41.0443, Z -7.1667, A 0.000, B 0.000, C 0.000 }
gfCNCPoint5[16398] = {X 73.8434, Y 41.6797, Z -7.1667, A 0.000, B 0.000, C 0.000 }
gfCNCPoint5[16399] = {X 74.3352, Y 42.4462, Z -7.1667, A 0.000, B 0.000, C 0.000 }
gfCNCPoint5[16400] = {X 74.6408, Y 43.3041, Z -7.1667, A 0.000, B 0.000, C 0.000 }
gfCNCPoint5[16401] = {X 74.7445, Y 44.2089, Z -7.1667, A 0.000, B 0.000, C 0.000 }
gfCNCPoint5[16402] = {X 74.7445, Y 45.0000, Z -7.1667, A 0.000, B 0.000, C 0.000 }
gfCNCPoint5[16403] = {X 74.6442, Y 45.8901, Z -7.1667, A 0.000, B 0.000, C 0.000 }
gfCNCPoint5[16404] = {X 74.3483, Y 46.7355, Z -7.1667, A 0.000, B 0.000, C 0.000 }
gfCNCPoint5[16405] = {X 73.8718, Y 47.4940, Z -7.1667, A 0.000, B 0.000, C 0.000 }
gfCNCPoint5[16406] = {X 73.2384, Y 48.1273, Z -7.1667, A 0.000, B 0.000, C 0.000 }
gfCNCPoint5[16407] = {X 72.4800, Y 48.6039, Z -7.1667, A 0.000, B 0.000, C 0.000 }
gfCNCPoint5[16408] = {X 71.6345, Y 48.8997, Z -7.1667, A 0.000, B 0.000, C 0.000 }
gfCNCPoint5[16409] = {X 70.7445, Y 49.0000, Z -7.1667, A 0.000, B 0.000, C 0.000 }
gfCNCPoint5[16410] = {X 64.1851, Y 49.0000, Z -7.1667, A 0.000, B 0.000, C 0.000 }
gfCNCPoint5[16411] = {X 63.2951, Y 48.8997, Z -7.1667, A 0.000, B 0.000, C 0.000 }
gfCNCPoint5[16412] = {X 62.4496, Y 48.6039, Z -7.1667, A 0.000, B 0.000, C 0.000 }
gfCNCPoint5[16413] = {X 61.6912, Y 48.1273, Z -7.1667, A 0.000, B 0.000, C 0.000 }
gfCNCPoint5[16414] = {X 61.0578, Y 47.4940, Z -7.1667, A 0.000, B 0.000, C 0.000 }
gfCNCPoint5[16415] = {X 60.5813, Y 46.7355, Z -7.1667, A 0.000, B 0.000, C 0.000 }
gfCNCPoint5[16416] = {X 60.2854, Y 45.8901, Z -7.1667, A 0.000, B 0.000, C 0.000 }
gfCNCPoint5[16417] = {X 60.1851, Y 45.0000, Z -7.1667, A 0.000, B 0.000, C 0.000 }
gfCNCPoint5[16418] = {X 60.1855, Y 44.1538, Z -7.1667, A 0.000, B 0.000, C 0.000 }
gfCNCPoint5[16419] = {X 60.2746, Y 43.3674, Z -7.1667, A 0.000, B 0.000, C 0.000 }
gfCNCPoint5[16420] = {X 60.5168, Y 42.6140, Z -7.1667, A 0.000, B 0.000, C 0.000 }
gfCNCPoint5[16421] = {X 60.9025, Y 41.9231, Z -7.1667, A 0.000, B 0.000, C 0.000 }
gfCNCPoint5[16422] = {X 60.9792, Y 41.8179, Z -7.1667, A 0.000, B 0.000, C 0.000 }
gfCNCPoint5[16423] = {X 60.2302, Y 39.7692, Z -7.1667, A 0.000, B 0.000, C 0.000 }
gfCNCPoint5[16424] = {X 51.8430, Y 39.7692, Z -7.1667, A 0.000, B 0.000, C 0.000 }
gfCNCPoint5[16425] = {X 51.8430, Y 39.8038, Z -7.1667, A 0.000, B 0.000, C 0.000 }
gfCNCPoint5[16426] = {X 50.9819, Y 42.1174, Z -7.1667, A 0.000, B 0.000, C 0.000 }
gfCNCPoint5[16427] = {X 51.0730, Y 42.2725, Z -7.1667, A 0.000, B 0.000, C 0.000 }
gfCNCPoint5[16428] = {X 51.3481, Y 42.8867, Z -7.1667, A 0.000, B 0.000, C 0.000 }
gfCNCPoint5[16429] = {X 51.5163, Y 43.5383, Z -7.1667, A 0.000, B 0.000, C 0.000 }
gfCNCPoint5[16430] = {X 51.5729, Y 44.2089, Z -7.1667, A 0.000, B 0.000, C 0.000 }
gfCNCPoint5[16431] = {X 51.5729, Y 45.0000, Z -7.1667, A 0.000, B 0.000, C 0.000 }
gfCNCPoint5[16432] = {X 51.4726, Y 45.8901, Z -7.1667, A 0.000, B 0.000, C 0.000 }
gfCNCPoint5[16433] = {X 51.1768, Y 46.7355, Z -7.1667, A 0.000, B 0.000, C 0.000 }
gfCNCPoint5[16434] = {X 50.7003, Y 47.4940, Z -7.1667, A 0.000, B 0.000, C 0.000 }
gfCNCPoint5[16435] = {X 50.0669, Y 48.1273, Z -7.1667, A 0.000, B 0.000, C 0.000 }
gfCNCPoint5[16436] = {X 49.3085, Y 48.6039, Z -7.1667, A 0.000, B 0.000, C 0.000 }
gfCNCPoint5[16437] = {X 48.4630, Y 48.8997, Z -7.1667, A 0.000, B 0.000, C 0.000 }
gfCNCPoint5[16438] = {X 47.5729, Y 49.0000, Z -7.1667, A 0.000, B 0.000, C 0.000 }
gfCNCPoint5[16439] = {X 40.6393, Y 49.0000, Z -7.1667, A 0.000, B 0.000, C 0.000 }
gfCNCPoint5[16440] = {X 39.7492, Y 48.8997, Z -7.1667, A 0.000, B 0.000, C 0.000 }
gfCNCPoint5[16441] = {X 38.9038, Y 48.6039, Z -7.1667, A 0.000, B 0.000, C 0.000 }
gfCNCPoint5[16442] = {X 38.1453, Y 48.1273, Z -7.1667, A 0.000, B 0.000, C 0.000 }
gfCNCPoint5[16443] = {X 37.5120, Y 47.4940, Z -7.1667, A 0.000, B 0.000, C 0.000 }
gfCNCPoint5[16444] = {X 37.0354, Y 46.7355, Z -7.1667, A 0.000, B 0.000, C 0.000 }
gfCNCPoint5[16445] = {X 36.7396, Y 45.8901, Z -7.1667, A 0.000, B 0.000, C 0.000 }
gfCNCPoint5[16446] = {X 36.6393, Y 45.0000, Z -7.1667, A 0.000, B 0.000, C 0.000 }
gfCNCPoint5[16447] = {X 36.6397, Y 44.1538, Z -7.1667, A 0.000, B 0.000, C 0.000 }
gfCNCPoint5[16448] = {X 36.7563, Y 43.2485, Z -7.1667, A 0.000, B 0.000, C 0.000 }
gfCNCPoint5[16449] = {X 37.0751, Y 42.3932, Z -7.1667, A 0.000, B 0.000, C 0.000 }
gfCNCPoint5[16450] = {X 37.5795, Y 41.6325, Z -7.1667, A 0.000, B 0.000, C 0.000 }
gfCNCPoint5[16451] = {X 38.2432, Y 41.0059, Z -7.1667, A 0.000, B 0.000, C 0.000 }
gfCNCPoint5[16452] = {X 39.0317, Y 40.5461, Z -7.1667, A 0.000, B 0.000, C 0.000 }
gfCNCPoint5[16453] = {X 39.0822, Y 40.5243, Z -7.1667, A 0.000, B 0.000, C 0.000 }
gfCNCPoint5[16454] = {X 39.1330, Y 40.5032, Z -7.1667, A 0.000, B 0.000, C 0.000 }
gfCNCPoint5[16455] = {X 39.1661, Y 40.4817, Z -7.1667, A 0.000, B 0.000, C 0.000 }
gfCNCPoint5[16456] = {X 39.1888, Y 40.4494, Z -7.1667, A 0.000, B 0.000, C 0.000 }
gfCNCPoint5[16457] = {X 39.2127, Y 40.3957, Z -7.1667, A 0.000, B 0.000, C 0.000 }
gfCNCPoint5[16458] = {X 39.2366, Y 40.3420, Z -7.1667, A 0.000, B 0.000, C 0.000 }
gfCNCPoint5[16459] = {X 39.8250, Y 38.9500, Z -7.1667, A 0.000, B 0.000, C 0.000 }
gfCNCPoint5[16460] = {X 40.3642, Y 37.5383, Z -7.1667, A 0.000, B 0.000, C 0.000 }
gfCNCPoint5[16461] = {X 43.9475, Y 27.9190, Z -7.1667, A 0.000, B 0.000, C 0.000 }
gfCNCPoint5[16462] = {X 40.1242, Y 26.4948, Z -7.1667, A 0.000, B 0.000, C 0.000 }
gfCNCPoint5[16463] = {X 40.1242, Y 26.4948, Z -4.1667, A 0.000, B 0.000, C 0.000 }
gfCNCPoint5[16464] = {X 40.1242, Y 26.4948, Z 11.0000, A 0.000, B 0.000, C 0.000 }
gfCNCPoint5[16465] = {X 79.0218, Y 28.5910, Z 11.0000, A 0.000, B 0.000, C 0.000 }
gfCNCPoint5[16466] = {X 79.0218, Y 28.5910, Z -4.1667, A 0.000, B 0.000, C 0.000 }
gfCNCPoint5[16467] = {X 79.0218, Y 28.5910, Z -7.1667, A 0.000, B 0.000, C 0.000 }
gfCNCPoint5[16468] = {X 83.1018, Y 28.5910, Z -7.1667, A 0.000, B 0.000, C 0.000 }
gfCNCPoint5[16469] = {X 83.1017, Y 16.2734, Z -7.1667, A 0.000, B 0.000, C 0.000 }
gfCNCPoint5[16470] = {X 82.4635, Y 15.6023, Z -7.1667, A 0.000, B 0.000, C 0.000 }
gfCNCPoint5[16471] = {X 81.9830, Y 14.8106, Z -7.1667, A 0.000, B 0.000, C 0.000 }
gfCNCPoint5[16472] = {X 81.6823, Y 13.9347, Z -7.1667, A 0.000, B 0.000, C 0.000 }
gfCNCPoint5[16473] = {X 81.5752, Y 13.0148, Z -7.1667, A 0.000, B 0.000, C 0.000 }
gfCNCPoint5[16474] = {X 81.5751, Y 12.1868, Z -7.1667, A 0.000, B 0.000, C 0.000 }
gfCNCPoint5[16475] = {X 81.6834, Y 11.2255, Z -7.1667, A 0.000, B 0.000, C 0.000 }
gfCNCPoint5[16476] = {X 82.0029, Y 10.3124, Z -7.1667, A 0.000, B 0.000, C 0.000 }
gfCNCPoint5[16477] = {X 82.5176, Y 9.4933, Z -7.1667, A 0.000, B 0.000, C 0.000 }
gfCNCPoint5[16478] = {X 83.2016, Y 8.8093, Z -7.1667, A 0.000, B 0.000, C 0.000 }
gfCNCPoint5[16479] = {X 84.0207, Y 8.2946, Z -7.1667, A 0.000, B 0.000, C 0.000 }
gfCNCPoint5[16480] = {X 84.9338, Y 7.9751, Z -7.1667, A 0.000, B 0.000, C 0.000 }
gfCNCPoint5[16481] = {X 85.8951, Y 7.8668, Z -7.1667, A 0.000, B 0.000, C 0.000 }
gfCNCPoint5[16482] = {X 94.0497, Y 7.8668, Z -7.1667, A 0.000, B 0.000, C 0.000 }
gfCNCPoint5[16483] = {X 95.0110, Y 7.9751, Z -7.1667, A 0.000, B 0.000, C 0.000 }
gfCNCPoint5[16484] = {X 95.9240, Y 8.2946, Z -7.1667, A 0.000, B 0.000, C 0.000 }
gfCNCPoint5[16485] = {X 96.7431, Y 8.8093, Z -7.1667, A 0.000, B 0.000, C 0.000 }
gfCNCPoint5[16486] = {X 97.4272, Y 9.4933, Z -7.1667, A 0.000, B 0.000, C 0.000 }
gfCNCPoint5[16487] = {X 97.9419, Y 10.3124, Z -7.1667, A 0.000, B 0.000, C 0.000 }
gfCNCPoint5[16488] = {X 98.2614, Y 11.2255, Z -7.1667, A 0.000, B 0.000, C 0.000 }
gfCNCPoint5[16489] = {X 98.3697, Y 12.1868, Z -7.1667, A 0.000, B 0.000, C 0.000 }
gfCNCPoint5[16490] = {X 98.3697, Y 12.9782, Z -7.1667, A 0.000, B 0.000, C 0.000 }
gfCNCPoint5[16491] = {X 98.2968, Y 13.7677, Z -7.1667, A 0.000, B 0.000, C 0.000 }
gfCNCPoint5[16492] = {X 98.0808, Y 14.5305, Z -7.1667, A 0.000, B 0.000, C 0.000 }
gfCNCPoint5[16493] = {X 97.7291, Y 15.2410, Z -7.1667, A 0.000, B 0.000, C 0.000 }
gfCNCPoint5[16494] = {X 101.8771, Y 25.5239, Z -7.1667, A 0.000, B 0.000, C 0.000 }
gfCNCPoint5[16495] = {X 106.0161, Y 15.2208, Z -7.1667, A 0.000, B 0.000, C 0.000 }
gfCNCPoint5[16496] = {X 105.6759, Y 14.5281, Z -7.1667, A 0.000, B 0.000, C 0.000 }
gfCNCPoint5[16497] = {X 105.4645, Y 13.7859, Z -7.1667, A 0.000, B 0.000, C 0.000 }
gfCNCPoint5[16498] = {X 105.3885, Y 13.0179, Z -7.1667, A 0.000, B 0.000, C 0.000 }
gfCNCPoint5[16499] = {X 105.3883, Y 12.1868, Z -7.1667, A 0.000, B 0.000, C 0.000 }
gfCNCPoint5[16500] = {X 105.4966, Y 11.2255, Z -7.1667, A 0.000, B 0.000, C 0.000 }
gfCNCPoint5[16501] = {X 105.8161, Y 10.3124, Z -7.1667, A 0.000, B 0.000, C 0.000 }
gfCNCPoint5[16502] = {X 106.3308, Y 9.4933, Z -7.1667, A 0.000, B 0.000, C 0.000 }
gfCNCPoint5[16503] = {X 107.0148, Y 8.8093, Z -7.1667, A 0.000, B 0.000, C 0.000 }
gfCNCPoint5[16504] = {X 107.8339, Y 8.2946, Z -7.1667, A 0.000, B 0.000, C 0.000 }
gfCNCPoint5[16505] = {X 108.7470, Y 7.9751, Z -7.1667, A 0.000, B 0.000, C 0.000 }
gfCNCPoint5[16506] = {X 109.7083, Y 7.8668, Z -7.1667, A 0.000, B 0.000, C 0.000 }
gfCNCPoint5[16507] = {X 117.7916, Y 7.8668, Z -7.1667, A 0.000, B 0.000, C 0.000 }
gfCNCPoint5[16508] = {X 118.7529, Y 7.9751, Z -7.1667, A 0.000, B 0.000, C 0.000 }
gfCNCPoint5[16509] = {X 119.6660, Y 8.2946, Z -7.1667, A 0.000, B 0.000, C 0.000 }
gfCNCPoint5[16510] = {X 120.4851, Y 8.8093, Z -7.1667, A 0.000, B 0.000, C 0.000 }
gfCNCPoint5[16511] = {X 121.1691, Y 9.4933, Z -7.1667, A 0.000, B 0.000, C 0.000 }
gfCNCPoint5[16512] = {X 121.6838, Y 10.3124, Z -7.1667, A 0.000, B 0.000, C 0.000 }
gfCNCPoint5[16513] = {X 122.0033, Y 11.2255, Z -7.1667, A 0.000, B 0.000, C 0.000 }
gfCNCPoint5[16514] = {X 122.1116, Y 12.1868, Z -7.1667, A 0.000, B 0.000, C 0.000 }
gfCNCPoint5[16515] = {X 122.1116, Y 12.9782, Z -7.1667, A 0.000, B 0.000, C 0.000 }
gfCNCPoint5[16516] = {X 122.0103, Y 13.9078, Z -7.1667, A 0.000, B 0.000, C 0.000 }
gfCNCPoint5[16517] = {X 121.7114, Y 14.7939, Z -7.1667, A 0.000, B 0.000, C 0.000 }
gfCNCPoint5[16518] = {X 121.2288, Y 15.5949, Z -7.1667, A 0.000, B 0.000, C 0.000 }
gfCNCPoint5[16519] = {X 120.5851, Y 16.2732, Z -7.1667, A 0.000, B 0.000, C 0.000 }
gfCNCPoint5[16520] = {X 120.5850, Y 40.9147, Z -7.1667, A 0.000, B 0.000, C 0.000 }
gfCNCPoint5[16521] = {X 120.6228, Y 40.9459, Z -7.1667, A 0.000, B 0.000, C 0.000 }
gfCNCPoint5[16522] = {X 121.2459, Y 41.6146, Z -7.1667, A 0.000, B 0.000, C 0.000 }
gfCNCPoint5[16523] = {X 121.7144, Y 42.3994, Z -7.1667, A 0.000, B 0.000, C 0.000 }
gfCNCPoint5[16524] = {X 122.0073, Y 43.2653, Z -7.1667, A 0.000, B 0.000, C 0.000 }
gfCNCPoint5[16525] = {X 122.1114, Y 44.1734, Z -7.1667, A 0.000, B 0.000, C 0.000 }
gfCNCPoint5[16526] = {X 122.1116, Y 45.0000, Z -7.1667, A 0.000, B 0.000, C 0.000 }
gfCNCPoint5[16527] = {X 122.0033, Y 45.9613, Z -7.1667, A 0.000, B 0.000, C 0.000 }
gfCNCPoint5[16528] = {X 121.6838, Y 46.8744, Z -7.1667, A 0.000, B 0.000, C 0.000 }
gfCNCPoint5[16529] = {X 121.1691, Y 47.6935, Z -7.1667, A 0.000, B 0.000, C 0.000 }
gfCNCPoint5[16530] = {X 120.4851, Y 48.3775, Z -7.1667, A 0.000, B 0.000, C 0.000 }
gfCNCPoint5[16531] = {X 119.6660, Y 48.8922, Z -7.1667, A 0.000, B 0.000, C 0.000 }
gfCNCPoint5[16532] = {X 118.7529, Y 49.2117, Z -7.1667, A 0.000, B 0.000, C 0.000 }
gfCNCPoint5[16533] = {X 117.7916, Y 49.3200, Z -7.1667, A 0.000, B 0.000, C 0.000 }
gfCNCPoint5[16534] = {X 111.9185, Y 49.3200, Z -7.1667, A 0.000, B 0.000, C 0.000 }
gfCNCPoint5[16535] = {X 110.9619, Y 49.2128, Z -7.1667, A 0.000, B 0.000, C 0.000 }
gfCNCPoint5[16536] = {X 110.0529, Y 48.8964, Z -7.1667, A 0.000, B 0.000, C 0.000 }
gfCNCPoint5[16537] = {X 109.2365, Y 48.3866, Z -7.1667, A 0.000, B 0.000, C 0.000 }
gfCNCPoint5[16538] = {X 108.5532, Y 47.7087, Z -7.1667, A 0.000, B 0.000, C 0.000 }
gfCNCPoint5[16539] = {X 108.0369, Y 46.8963, Z -7.1667, A 0.000, B 0.000, C 0.000 }
gfCNCPoint5[16540] = {X 107.7134, Y 45.9898, Z -7.1667, A 0.000, B 0.000, C 0.000 }
gfCNCPoint5[16541] = {X 107.5986, Y 45.0341, Z -7.1667, A 0.000, B 0.000, C 0.000 }
gfCNCPoint5[16542] = {X 107.5985, Y 44.1771, Z -7.1667, A 0.000, B 0.000, C 0.000 }
gfCNCPoint5[16543] = {X 107.6338, Y 43.6368, Z -7.1667, A 0.000, B 0.000, C 0.000 }
gfCNCPoint5[16544] = {X 107.7391, Y 43.1057, Z -7.1667, A 0.000, B 0.000, C 0.000 }
gfCNCPoint5[16545] = {X 107.9078, Y 42.6046, Z -7.1667, A 0.000, B 0.000, C 0.000 }
gfCNCPoint5[16546] = {X 108.1388, Y 42.1290, Z -7.1667, A 0.000, B 0.000, C 0.000 }
gfCNCPoint5[16547] = {X 108.5880, Y 41.4615, Z -7.1667, A 0.000, B 0.000, C 0.000 }
gfCNCPoint5[16548] = {X 109.1249, Y 40.8623, Z -7.1667, A 0.000, B 0.000, C 0.000 }
gfCNCPoint5[16549] = {X 109.1248, Y 39.2986, Z -7.1667, A 0.000, B 0.000, C 0.000 }
gfCNCPoint5[16550] = {X 106.1118, Y 46.6615, Z -7.1667, A 0.000, B 0.000, C 0.000 }
gfCNCPoint5[16551] = {X 105.7417, Y 47.3611, Z -7.1667, A 0.000, B 0.000, C 0.000 }
gfCNCPoint5[16552] = {X 105.2502, Y 47.9815, Z -7.1667, A 0.000, B 0.000, C 0.000 }
gfCNCPoint5[16553] = {X 104.6538, Y 48.5018, Z -7.1667, A 0.000, B 0.000, C 0.000 }
gfCNCPoint5[16554] = {X 103.9724, Y 48.9046, Z -7.1667, A 0.000, B 0.000, C 0.000 }
gfCNCPoint5[16555] = {X 103.0287, Y 49.2242, Z -7.1667, A 0.000, B 0.000, C 0.000 }
gfCNCPoint5[16556] = {X 102.0368, Y 49.3191, Z -7.1667, A 0.000, B 0.000, C 0.000 }
gfCNCPoint5[16557] = {X 101.0496, Y 49.1842, Z -7.1667, A 0.000, B 0.000, C 0.000 }
gfCNCPoint5[16558] = {X 100.1195, Y 48.8268, Z -7.1667, A 0.000, B 0.000, C 0.000 }
gfCNCPoint5[16559] = {X 99.2961, Y 48.2657, Z -7.1667, A 0.000, B 0.000, C 0.000 }
gfCNCPoint5[16560] = {X 98.6231, Y 47.5309, Z -7.1667, A 0.000, B 0.000, C 0.000 }
gfCNCPoint5[16561] = {X 98.1363, Y 46.6615, Z -7.1667, A 0.000, B 0.000, C 0.000 }
gfCNCPoint5[16562] = {X 95.1320, Y 39.3141, Z -7.1667, A 0.000, B 0.000, C 0.000 }
gfCNCPoint5[16563] = {X 95.1320, Y 40.9046, Z -7.1667, A 0.000, B 0.000, C 0.000 }
gfCNCPoint5[16564] = {X 95.6571, Y 41.4420, Z -7.1667, A 0.000, B 0.000, C 0.000 }
gfCNCPoint5[16565] = {X 96.0830, Y 42.0609, Z -7.1667, A 0.000, B 0.000, C 0.000 }
gfCNCPoint5[16566] = {X 96.3314, Y 42.5715, Z -7.1667, A 0.000, B 0.000, C 0.000 }
gfCNCPoint5[16567] = {X 96.5119, Y 43.1099, Z -7.1667, A 0.000, B 0.000, C 0.000 }
gfCNCPoint5[16568] = {X 96.6198, Y 43.6537, Z -7.1667, A 0.000, B 0.000, C 0.000 }
gfCNCPoint5[16569] = {X 96.6585, Y 44.2067, Z -7.1667, A 0.000, B 0.000, C 0.000 }
gfCNCPoint5[16570] = {X 96.6583, Y 45.0415, Z -7.1667, A 0.000, B 0.000, C 0.000 }
gfCNCPoint5[16571] = {X 96.5422, Y 45.9960, Z -7.1667, A 0.000, B 0.000, C 0.000 }
gfCNCPoint5[16572] = {X 96.2178, Y 46.9011, Z -7.1667, A 0.000, B 0.000, C 0.000 }
gfCNCPoint5[16573] = {X 95.7012, Y 47.7120, Z -7.1667, A 0.000, B 0.000, C 0.000 }
gfCNCPoint5[16574] = {X 95.0181, Y 48.3886, Z -7.1667, A 0.000, B 0.000, C 0.000 }
gfCNCPoint5[16575] = {X 94.2022, Y 48.8973, Z -7.1667, A 0.000, B 0.000, C 0.000 }
gfCNCPoint5[16576] = {X 93.2940, Y 49.2130, Z -7.1667, A 0.000, B 0.000, C 0.000 }
gfCNCPoint5[16577] = {X 92.3385, Y 49.3200, Z -7.1667, A 0.000, B 0.000, C 0.000 }
gfCNCPoint5[16578] = {X 85.8951, Y 49.3200, Z -7.1667, A 0.000, B 0.000, C 0.000 }
gfCNCPoint5[16579] = {X 84.9387, Y 49.2128, Z -7.1667, A 0.000, B 0.000, C 0.000 }
gfCNCPoint5[16580] = {X 84.0297, Y 48.8965, Z -7.1667, A 0.000, B 0.000, C 0.000 }
gfCNCPoint5[16581] = {X 83.2134, Y 48.3869, Z -7.1667, A 0.000, B 0.000, C 0.000 }
gfCNCPoint5[16582] = {X 82.5301, Y 47.7091, Z -7.1667, A 0.000, B 0.000, C 0.000 }
gfCNCPoint5[16583] = {X 82.0138, Y 46.8970, Z -7.1667, A 0.000, B 0.000, C 0.000 }
gfCNCPoint5[16584] = {X 81.6902, Y 45.9906, Z -7.1667, A 0.000, B 0.000, C 0.000 }
gfCNCPoint5[16585] = {X 81.5752, Y 45.0351, Z -7.1667, A 0.000, B 0.000, C 0.000 }
gfCNCPoint5[16586] = {X 81.5751, Y 44.2072, Z -7.1667, A 0.000, B 0.000, C 0.000 }
gfCNCPoint5[16587] = {X 81.6798, Y 43.2778, Z -7.1667, A 0.000, B 0.000, C 0.000 }
gfCNCPoint5[16588] = {X 81.9796, Y 42.3918, Z -7.1667, A 0.000, B 0.000, C 0.000 }
gfCNCPoint5[16589] = {X 82.4610, Y 41.5899, Z -7.1667, A 0.000, B 0.000, C 0.000 }
gfCNCPoint5[16590] = {X 83.1019, Y 40.9086, Z -7.1667, A 0.000, B 0.000, C 0.000 }
gfCNCPoint5[16591] = {X 83.1018, Y 28.5910, Z -7.1667, A 0.000, B 0.000, C 0.000 }
gfCNCPoint5[16592] = {X 79.1018, Y 28.5910, Z -7.1667, A 0.000, B 0.000, C 0.000 }
gfCNCPoint5[16593] = {X 83.1818, Y 28.5910, Z -7.1667, A 0.000, B 0.000, C 0.000 }
gfCNCPoint5[16594] = {X 83.1817, Y 16.2361, Z -7.1667, A 0.000, B 0.000, C 0.000 }
gfCNCPoint5[16595] = {X 82.5440, Y 15.5756, Z -7.1667, A 0.000, B 0.000, C 0.000 }
gfCNCPoint5[16596] = {X 82.0633, Y 14.7934, Z -7.1667, A 0.000, B 0.000, C 0.000 }
gfCNCPoint5[16597] = {X 81.7624, Y 13.9260, Z -7.1667, A 0.000, B 0.000, C 0.000 }
gfCNCPoint5[16598] = {X 81.6552, Y 13.0142, Z -7.1667, A 0.000, B 0.000, C 0.000 }
gfCNCPoint5[16599] = {X 81.6551, Y 12.1868, Z -7.1667, A 0.000, B 0.000, C 0.000 }
gfCNCPoint5[16600] = {X 81.7614, Y 11.2433, Z -7.1667, A 0.000, B 0.000, C 0.000 }
gfCNCPoint5[16601] = {X 82.0750, Y 10.3472, Z -7.1667, A 0.000, B 0.000, C 0.000 }
gfCNCPoint5[16602] = {X 82.5801, Y 9.5432, Z -7.1667, A 0.000, B 0.000, C 0.000 }
gfCNCPoint5[16603] = {X 83.2515, Y 8.8719, Z -7.1667, A 0.000, B 0.000, C 0.000 }
gfCNCPoint5[16604] = {X 84.0554, Y 8.3667, Z -7.1667, A 0.000, B 0.000, C 0.000 }
gfCNCPoint5[16605] = {X 84.9516, Y 8.0531, Z -7.1667, A 0.000, B 0.000, C 0.000 }
gfCNCPoint5[16606] = {X 85.8951, Y 7.9468, Z -7.1667, A 0.000, B 0.000, C 0.000 }
gfCNCPoint5[16607] = {X 94.0497, Y 7.9468, Z -7.1667, A 0.000, B 0.000, C 0.000 }
gfCNCPoint5[16608] = {X 94.9932, Y 8.0531, Z -7.1667, A 0.000, B 0.000, C 0.000 }
gfCNCPoint5[16609] = {X 95.8893, Y 8.3667, Z -7.1667, A 0.000, B 0.000, C 0.000 }
gfCNCPoint5[16610] = {X 96.6933, Y 8.8718, Z -7.1667, A 0.000, B 0.000, C 0.000 }
gfCNCPoint5[16611] = {X 97.3646, Y 9.5432, Z -7.1667, A 0.000, B 0.000, C 0.000 }
gfCNCPoint5[16612] = {X 97.8698, Y 10.3471, Z -7.1667, A 0.000, B 0.000, C 0.000 }
gfCNCPoint5[16613] = {X 98.1834, Y 11.2433, Z -7.1667, A 0.000, B 0.000, C 0.000 }
gfCNCPoint5[16614] = {X 98.2897, Y 12.1868, Z -7.1667, A 0.000, B 0.000, C 0.000 }
gfCNCPoint5[16615] = {X 98.2897, Y 12.9782, Z -7.1667, A 0.000, B 0.000, C 0.000 }
gfCNCPoint5[16616] = {X 98.2156, Y 13.7662, Z -7.1667, A 0.000, B 0.000, C 0.000 }
gfCNCPoint5[16617] = {X 97.9964, Y 14.5267, Z -7.1667, A 0.000, B 0.000, C 0.000 }
gfCNCPoint5[16618] = {X 97.6397, Y 15.2333, Z -7.1667, A 0.000, B 0.000, C 0.000 }
gfCNCPoint5[16619] = {X 101.8773, Y 25.7381, Z -7.1667, A 0.000, B 0.000, C 0.000 }
gfCNCPoint5[16620] = {X 106.1053, Y 15.2133, Z -7.1667, A 0.000, B 0.000, C 0.000 }
gfCNCPoint5[16621] = {X 105.7602, Y 14.5242, Z -7.1667, A 0.000, B 0.000, C 0.000 }
gfCNCPoint5[16622] = {X 105.5456, Y 13.7840, Z -7.1667, A 0.000, B 0.000, C 0.000 }
gfCNCPoint5[16623] = {X 105.4685, Y 13.0172, Z -7.1667, A 0.000, B 0.000, C 0.000 }
gfCNCPoint5[16624] = {X 105.4683, Y 12.1868, Z -7.1667, A 0.000, B 0.000, C 0.000 }
gfCNCPoint5[16625] = {X 105.5746, Y 11.2433, Z -7.1667, A 0.000, B 0.000, C 0.000 }
gfCNCPoint5[16626] = {X 105.8882, Y 10.3471, Z -7.1667, A 0.000, B 0.000, C 0.000 }
gfCNCPoint5[16627] = {X 106.3933, Y 9.5432, Z -7.1667, A 0.000, B 0.000, C 0.000 }
gfCNCPoint5[16628] = {X 107.0647, Y 8.8718, Z -7.1667, A 0.000, B 0.000, C 0.000 }
gfCNCPoint5[16629] = {X 107.8686, Y 8.3667, Z -7.1667, A 0.000, B 0.000, C 0.000 }
gfCNCPoint5[16630] = {X 108.7648, Y 8.0531, Z -7.1667, A 0.000, B 0.000, C 0.000 }
gfCNCPoint5[16631] = {X 109.7083, Y 7.9468, Z -7.1667, A 0.000, B 0.000, C 0.000 }
gfCNCPoint5[16632] = {X 117.7916, Y 7.9468, Z -7.1667, A 0.000, B 0.000, C 0.000 }
gfCNCPoint5[16633] = {X 118.7351, Y 8.0531, Z -7.1667, A 0.000, B 0.000, C 0.000 }
gfCNCPoint5[16634] = {X 119.6312, Y 8.3667, Z -7.1667, A 0.000, B 0.000, C 0.000 }
gfCNCPoint5[16635] = {X 120.4352, Y 8.8718, Z -7.1667, A 0.000, B 0.000, C 0.000 }
gfCNCPoint5[16636] = {X 121.1065, Y 9.5432, Z -7.1667, A 0.000, B 0.000, C 0.000 }
gfCNCPoint5[16637] = {X 121.6117, Y 10.3471, Z -7.1667, A 0.000, B 0.000, C 0.000 }
gfCNCPoint5[16638] = {X 121.9253, Y 11.2433, Z -7.1667, A 0.000, B 0.000, C 0.000 }
gfCNCPoint5[16639] = {X 122.0316, Y 12.1868, Z -7.1667, A 0.000, B 0.000, C 0.000 }
gfCNCPoint5[16640] = {X 122.0316, Y 12.9782, Z -7.1667, A 0.000, B 0.000, C 0.000 }
gfCNCPoint5[16641] = {X 121.9302, Y 13.8996, Z -7.1667, A 0.000, B 0.000, C 0.000 }
gfCNCPoint5[16642] = {X 121.6310, Y 14.7770, Z -7.1667, A 0.000, B 0.000, C 0.000 }
gfCNCPoint5[16643] = {X 121.1483, Y 15.5684, Z -7.1667, A 0.000, B 0.000, C 0.000 }
gfCNCPoint5[16644] = {X 120.5051, Y 16.2360, Z -7.1667, A 0.000, B 0.000, C 0.000 }
gfCNCPoint5[16645] = {X 120.5050, Y 40.9524, Z -7.1667, A 0.000, B 0.000, C 0.000 }
gfCNCPoint5[16646] = {X 120.5711, Y 41.0070, Z -7.1667, A 0.000, B 0.000, C 0.000 }
gfCNCPoint5[16647] = {X 121.1824, Y 41.6632, Z -7.1667, A 0.000, B 0.000, C 0.000 }
gfCNCPoint5[16648] = {X 121.6420, Y 42.4334, Z -7.1667, A 0.000, B 0.000, C 0.000 }
gfCNCPoint5[16649] = {X 121.9293, Y 43.2830, Z -7.1667, A 0.000, B 0.000, C 0.000 }
gfCNCPoint5[16650] = {X 122.0314, Y 44.1740, Z -7.1667, A 0.000, B 0.000, C 0.000 }
gfCNCPoint5[16651] = {X 122.0316, Y 45.0000, Z -7.1667, A 0.000, B 0.000, C 0.000 }
gfCNCPoint5[16652] = {X 121.9253, Y 45.9435, Z -7.1667, A 0.000, B 0.000, C 0.000 }
gfCNCPoint5[16653] = {X 121.6117, Y 46.8397, Z -7.1667, A 0.000, B 0.000, C 0.000 }
gfCNCPoint5[16654] = {X 121.1065, Y 47.6436, Z -7.1667, A 0.000, B 0.000, C 0.000 }
gfCNCPoint5[16655] = {X 120.4352, Y 48.3150, Z -7.1667, A 0.000, B 0.000, C 0.000 }
gfCNCPoint5[16656] = {X 119.6312, Y 48.8201, Z -7.1667, A 0.000, B 0.000, C 0.000 }
gfCNCPoint5[16657] = {X 118.7351, Y 49.1337, Z -7.1667, A 0.000, B 0.000, C 0.000 }
gfCNCPoint5[16658] = {X 117.7916, Y 49.2400, Z -7.1667, A 0.000, B 0.000, C 0.000 }
gfCNCPoint5[16659] = {X 111.9185, Y 49.2400, Z -7.1667, A 0.000, B 0.000, C 0.000 }
gfCNCPoint5[16660] = {X 110.9797, Y 49.1348, Z -7.1667, A 0.000, B 0.000, C 0.000 }
gfCNCPoint5[16661] = {X 110.0874, Y 48.8242, Z -7.1667, A 0.000, B 0.000, C 0.000 }
gfCNCPoint5[16662] = {X 109.2861, Y 48.3239, Z -7.1667, A 0.000, B 0.000, C 0.000 }
gfCNCPoint5[16663] = {X 108.6155, Y 47.6585, Z -7.1667, A 0.000, B 0.000, C 0.000 }
gfCNCPoint5[16664] = {X 108.1088, Y 46.8612, Z -7.1667, A 0.000, B 0.000, C 0.000 }
gfCNCPoint5[16665] = {X 107.7913, Y 45.9714, Z -7.1667, A 0.000, B 0.000, C 0.000 }
gfCNCPoint5[16666] = {X 107.6786, Y 45.0335, Z -7.1667, A 0.000, B 0.000, C 0.000 }
gfCNCPoint5[16667] = {X 107.6785, Y 44.1771, Z -7.1667, A 0.000, B 0.000, C 0.000 }
gfCNCPoint5[16668] = {X 107.7131, Y 43.6472, Z -7.1667, A 0.000, B 0.000, C 0.000 }
gfCNCPoint5[16669] = {X 107.8164, Y 43.1264, Z -7.1667, A 0.000, B 0.000, C 0.000 }
gfCNCPoint5[16670] = {X 107.9818, Y 42.6349, Z -7.1667, A 0.000, B 0.000, C 0.000 }
gfCNCPoint5[16671] = {X 108.2084, Y 42.1685, Z -7.1667, A 0.000, B 0.000, C 0.000 }
gfCNCPoint5[16672] = {X 108.6616, Y 41.4971, Z -7.1667, A 0.000, B 0.000, C 0.000 }
gfCNCPoint5[16673] = {X 109.2049, Y 40.8963, Z -7.1667, A 0.000, B 0.000, C 0.000 }
gfCNCPoint5[16674] = {X 109.2048, Y 39.1629, Z -7.1667, A 0.000, B 0.000, C 0.000 }
gfCNCPoint5[16675] = {X 109.0939, Y 39.1629, Z -7.1667, A 0.000, B 0.000, C 0.000 }
gfCNCPoint5[16676] = {X 106.0379, Y 46.6307, Z -7.1667, A 0.000, B 0.000, C 0.000 }
gfCNCPoint5[16677] = {X 105.6747, Y 47.3174, Z -7.1667, A 0.000, B 0.000, C 0.000 }
gfCNCPoint5[16678] = {X 105.1923, Y 47.9263, Z -7.1667, A 0.000, B 0.000, C 0.000 }
gfCNCPoint5[16679] = {X 104.6069, Y 48.4370, Z -7.1667, A 0.000, B 0.000, C 0.000 }
gfCNCPoint5[16680] = {X 103.9382, Y 48.8323, Z -7.1667, A 0.000, B 0.000, C 0.000 }
gfCNCPoint5[16681] = {X 103.0119, Y 49.1460, Z -7.1667, A 0.000, B 0.000, C 0.000 }
gfCNCPoint5[16682] = {X 102.0384, Y 49.2391, Z -7.1667, A 0.000, B 0.000, C 0.000 }
gfCNCPoint5[16683] = {X 101.0695, Y 49.1068, Z -7.1667, A 0.000, B 0.000, C 0.000 }
gfCNCPoint5[16684] = {X 100.1566, Y 48.7559, Z -7.1667, A 0.000, B 0.000, C 0.000 }
gfCNCPoint5[16685] = {X 99.3484, Y 48.2052, Z -7.1667, A 0.000, B 0.000, C 0.000 }
gfCNCPoint5[16686] = {X 98.6879, Y 47.4840, Z -7.1667, A 0.000, B 0.000, C 0.000 }
gfCNCPoint5[16687] = {X 98.2102, Y 46.6307, Z -7.1667, A 0.000, B 0.000, C 0.000 }
gfCNCPoint5[16688] = {X 95.0520, Y 38.9070, Z -7.1667, A 0.000, B 0.000, C 0.000 }
gfCNCPoint5[16689] = {X 95.0520, Y 40.9415, Z -7.1667, A 0.000, B 0.000, C 0.000 }
gfCNCPoint5[16690] = {X 95.5836, Y 41.4788, Z -7.1667, A 0.000, B 0.000, C 0.000 }
gfCNCPoint5[16691] = {X 96.0135, Y 42.1005, Z -7.1667, A 0.000, B 0.000, C 0.000 }
gfCNCPoint5[16692] = {X 96.2573, Y 42.6018, Z -7.1667, A 0.000, B 0.000, C 0.000 }
gfCNCPoint5[16693] = {X 96.4346, Y 43.1304, Z -7.1667, A 0.000, B 0.000, C 0.000 }
gfCNCPoint5[16694] = {X 96.5405, Y 43.6643, Z -7.1667, A 0.000, B 0.000, C 0.000 }
gfCNCPoint5[16695] = {X 96.5785, Y 44.2072, Z -7.1667, A 0.000, B 0.000, C 0.000 }
gfCNCPoint5[16696] = {X 96.5783, Y 45.0408, Z -7.1667, A 0.000, B 0.000, C 0.000 }
gfCNCPoint5[16697] = {X 96.4643, Y 45.9775, Z -7.1667, A 0.000, B 0.000, C 0.000 }
gfCNCPoint5[16698] = {X 96.1459, Y 46.8659, Z -7.1667, A 0.000, B 0.000, C 0.000 }
gfCNCPoint5[16699] = {X 95.6389, Y 47.6618, Z -7.1667, A 0.000, B 0.000, C 0.000 }
gfCNCPoint5[16700] = {X 94.9685, Y 48.3258, Z -7.1667, A 0.000, B 0.000, C 0.000 }
gfCNCPoint5[16701] = {X 94.1677, Y 48.8251, Z -7.1667, A 0.000, B 0.000, C 0.000 }
gfCNCPoint5[16702] = {X 93.2764, Y 49.1350, Z -7.1667, A 0.000, B 0.000, C 0.000 }
gfCNCPoint5[16703] = {X 92.3385, Y 49.2400, Z -7.1667, A 0.000, B 0.000, C 0.000 }
gfCNCPoint5[16704] = {X 85.8951, Y 49.2400, Z -7.1667, A 0.000, B 0.000, C 0.000 }
gfCNCPoint5[16705] = {X 84.9564, Y 49.1348, Z -7.1667, A 0.000, B 0.000, C 0.000 }
gfCNCPoint5[16706] = {X 84.0643, Y 48.8244, Z -7.1667, A 0.000, B 0.000, C 0.000 }
gfCNCPoint5[16707] = {X 83.2631, Y 48.3242, Z -7.1667, A 0.000, B 0.000, C 0.000 }
gfCNCPoint5[16708] = {X 82.5924, Y 47.6590, Z -7.1667, A 0.000, B 0.000, C 0.000 }
gfCNCPoint5[16709] = {X 82.0857, Y 46.8618, Z -7.1667, A 0.000, B 0.000, C 0.000 }
gfCNCPoint5[16710] = {X 81.7681, Y 45.9723, Z -7.1667, A 0.000, B 0.000, C 0.000 }
gfCNCPoint5[16711] = {X 81.6552, Y 45.0345, Z -7.1667, A 0.000, B 0.000, C 0.000 }
gfCNCPoint5[16712] = {X 81.6551, Y 44.2076, Z -7.1667, A 0.000, B 0.000, C 0.000 }
gfCNCPoint5[16713] = {X 81.7598, Y 43.2862, Z -7.1667, A 0.000, B 0.000, C 0.000 }
gfCNCPoint5[16714] = {X 82.0600, Y 42.4088, Z -7.1667, A 0.000, B 0.000, C 0.000 }
gfCNCPoint5[16715] = {X 82.5415, Y 41.6163, Z -7.1667, A 0.000, B 0.000, C 0.000 }
gfCNCPoint5[16716] = {X 83.1819, Y 40.9456, Z -7.1667, A 0.000, B 0.000, C 0.000 }
gfCNCPoint5[16717] = {X 83.1818, Y 28.5910, Z -7.1667, A 0.000, B 0.000, C 0.000 }
gfCNCPoint5[16718] = {X 79.1818, Y 28.5910, Z -7.1667, A 0.000, B 0.000, C 0.000 }
gfCNCPoint5[16719] = {X 83.2618, Y 28.5910, Z -7.1667, A 0.000, B 0.000, C 0.000 }
gfCNCPoint5[16720] = {X 83.2617, Y 16.1984, Z -7.1667, A 0.000, B 0.000, C 0.000 }
gfCNCPoint5[16721] = {X 82.6244, Y 15.5487, Z -7.1667, A 0.000, B 0.000, C 0.000 }
gfCNCPoint5[16722] = {X 82.1437, Y 14.7760, Z -7.1667, A 0.000, B 0.000, C 0.000 }
gfCNCPoint5[16723] = {X 81.8425, Y 13.9172, Z -7.1667, A 0.000, B 0.000, C 0.000 }
gfCNCPoint5[16724] = {X 81.7352, Y 13.0135, Z -7.1667, A 0.000, B 0.000, C 0.000 }
gfCNCPoint5[16725] = {X 81.7351, Y 12.1868, Z -7.1667, A 0.000, B 0.000, C 0.000 }
gfCNCPoint5[16726] = {X 81.8394, Y 11.2611, Z -7.1667, A 0.000, B 0.000, C 0.000 }
gfCNCPoint5[16727] = {X 82.1470, Y 10.3819, Z -7.1667, A 0.000, B 0.000, C 0.000 }
gfCNCPoint5[16728] = {X 82.6427, Y 9.5931, Z -7.1667, A 0.000, B 0.000, C 0.000 }
gfCNCPoint5[16729] = {X 83.3014, Y 8.9344, Z -7.1667, A 0.000, B 0.000, C 0.000 }
gfCNCPoint5[16730] = {X 84.0901, Y 8.4388, Z -7.1667, A 0.000, B 0.000, C 0.000 }
gfCNCPoint5[16731] = {X 84.9694, Y 8.1311, Z -7.1667, A 0.000, B 0.000, C 0.000 }
gfCNCPoint5[16732] = {X 85.8951, Y 8.0268, Z -7.1667, A 0.000, B 0.000, C 0.000 }
gfCNCPoint5[16733] = {X 94.0497, Y 8.0268, Z -7.1667, A 0.000, B 0.000, C 0.000 }
gfCNCPoint5[16734] = {X 94.9754, Y 8.1311, Z -7.1667, A 0.000, B 0.000, C 0.000 }
gfCNCPoint5[16735] = {X 95.8546, Y 8.4388, Z -7.1667, A 0.000, B 0.000, C 0.000 }
gfCNCPoint5[16736] = {X 96.6434, Y 8.9344, Z -7.1667, A 0.000, B 0.000, C 0.000 }
gfCNCPoint5[16737] = {X 97.3021, Y 9.5931, Z -7.1667, A 0.000, B 0.000, C 0.000 }
gfCNCPoint5[16738] = {X 97.7977, Y 10.3819, Z -7.1667, A 0.000, B 0.000, C 0.000 }
gfCNCPoint5[16739] = {X 98.1054, Y 11.2611, Z -7.1667, A 0.000, B 0.000, C 0.000 }
gfCNCPoint5[16740] = {X 98.2097, Y 12.1868, Z -7.1667, A 0.000, B 0.000, C 0.000 }
gfCNCPoint5[16741] = {X 98.2097, Y 12.9782, Z -7.1667, A 0.000, B 0.000, C 0.000 }
gfCNCPoint5[16742] = {X 98.1344, Y 13.7657, Z -7.1667, A 0.000, B 0.000, C 0.000 }
gfCNCPoint5[16743] = {X 97.9115, Y 14.5247, Z -7.1667, A 0.000, B 0.000, C 0.000 }
gfCNCPoint5[16744] = {X 97.5489, Y 15.2277, Z -7.1667, A 0.000, B 0.000, C 0.000 }
gfCNCPoint5[16745] = {X 101.8774, Y 25.9524, Z -7.1667, A 0.000, B 0.000, C 0.000 }
gfCNCPoint5[16746] = {X 106.1948, Y 15.2053, Z -7.1667, A 0.000, B 0.000, C 0.000 }
gfCNCPoint5[16747] = {X 105.8446, Y 14.5200, Z -7.1667, A 0.000, B 0.000, C 0.000 }
gfCNCPoint5[16748] = {X 105.6267, Y 13.7820, Z -7.1667, A 0.000, B 0.000, C 0.000 }
gfCNCPoint5[16749] = {X 105.5485, Y 13.0164, Z -7.1667, A 0.000, B 0.000, C 0.000 }
gfCNCPoint5[16750] = {X 105.5483, Y 12.1868, Z -7.1667, A 0.000, B 0.000, C 0.000 }
gfCNCPoint5[16751] = {X 105.6526, Y 11.2611, Z -7.1667, A 0.000, B 0.000, C 0.000 }
gfCNCPoint5[16752] = {X 105.9602, Y 10.3819, Z -7.1667, A 0.000, B 0.000, C 0.000 }
gfCNCPoint5[16753] = {X 106.4559, Y 9.5931, Z -7.1667, A 0.000, B 0.000, C 0.000 }
gfCNCPoint5[16754] = {X 107.1146, Y 8.9344, Z -7.1667, A 0.000, B 0.000, C 0.000 }
gfCNCPoint5[16755] = {X 107.9033, Y 8.4388, Z -7.1667, A 0.000, B 0.000, C 0.000 }
gfCNCPoint5[16756] = {X 108.7826, Y 8.1311, Z -7.1667, A 0.000, B 0.000, C 0.000 }
gfCNCPoint5[16757] = {X 109.7083, Y 8.0268, Z -7.1667, A 0.000, B 0.000, C 0.000 }
gfCNCPoint5[16758] = {X 117.7916, Y 8.0268, Z -7.1667, A 0.000, B 0.000, C 0.000 }
gfCNCPoint5[16759] = {X 118.7173, Y 8.1311, Z -7.1667, A 0.000, B 0.000, C 0.000 }
gfCNCPoint5[16760] = {X 119.5965, Y 8.4388, Z -7.1667, A 0.000, B 0.000, C 0.000 }
gfCNCPoint5[16761] = {X 120.3853, Y 8.9344, Z -7.1667, A 0.000, B 0.000, C 0.000 }
gfCNCPoint5[16762] = {X 121.0440, Y 9.5931, Z -7.1667, A 0.000, B 0.000, C 0.000 }
gfCNCPoint5[16763] = {X 121.5396, Y 10.3819, Z -7.1667, A 0.000, B 0.000, C 0.000 }
gfCNCPoint5[16764] = {X 121.8473, Y 11.2611, Z -7.1667, A 0.000, B 0.000, C 0.000 }
gfCNCPoint5[16765] = {X 121.9516, Y 12.1868, Z -7.1667, A 0.000, B 0.000, C 0.000 }
gfCNCPoint5[16766] = {X 121.9516, Y 12.9782, Z -7.1667, A 0.000, B 0.000, C 0.000 }
gfCNCPoint5[16767] = {X 121.8501, Y 13.8913, Z -7.1667, A 0.000, B 0.000, C 0.000 }
gfCNCPoint5[16768] = {X 121.5506, Y 14.7599, Z -7.1667, A 0.000, B 0.000, C 0.000 }
gfCNCPoint5[16769] = {X 121.0678, Y 15.5416, Z -7.1667, A 0.000, B 0.000, C 0.000 }
gfCNCPoint5[16770] = {X 120.4251, Y 16.1983, Z -7.1667, A 0.000, B 0.000, C 0.000 }
gfCNCPoint5[16771] = {X 120.4250, Y 40.9901, Z -7.1667, A 0.000, B 0.000, C 0.000 }
gfCNCPoint5[16772] = {X 120.5194, Y 41.0680, Z -7.1667, A 0.000, B 0.000, C 0.000 }
gfCNCPoint5[16773] = {X 121.1189, Y 41.7119, Z -7.1667, A 0.000, B 0.000, C 0.000 }
gfCNCPoint5[16774] = {X 121.5695, Y 42.4673, Z -7.1667, A 0.000, B 0.000, C 0.000 }
gfCNCPoint5[16775] = {X 121.8513, Y 43.3007, Z -7.1667, A 0.000, B 0.000, C 0.000 }
gfCNCPoint5[16776] = {X 121.9514, Y 44.1747, Z -7.1667, A 0.000, B 0.000, C 0.000 }
gfCNCPoint5[16777] = {X 121.9516, Y 45.0000, Z -7.1667, A 0.000, B 0.000, C 0.000 }
gfCNCPoint5[16778] = {X 121.8473, Y 45.9257, Z -7.1667, A 0.000, B 0.000, C 0.000 }
gfCNCPoint5[16779] = {X 121.5396, Y 46.8050, Z -7.1667, A 0.000, B 0.000, C 0.000 }
gfCNCPoint5[16780] = {X 121.0440, Y 47.5937, Z -7.1667, A 0.000, B 0.000, C 0.000 }
gfCNCPoint5[16781] = {X 120.3853, Y 48.2524, Z -7.1667, A 0.000, B 0.000, C 0.000 }
gfCNCPoint5[16782] = {X 119.5965, Y 48.7480, Z -7.1667, A 0.000, B 0.000, C 0.000 }
gfCNCPoint5[16783] = {X 118.7173, Y 49.0557, Z -7.1667, A 0.000, B 0.000, C 0.000 }
gfCNCPoint5[16784] = {X 117.7916, Y 49.1600, Z -7.1667, A 0.000, B 0.000, C 0.000 }
gfCNCPoint5[16785] = {X 111.9185, Y 49.1600, Z -7.1667, A 0.000, B 0.000, C 0.000 }
gfCNCPoint5[16786] = {X 110.9974, Y 49.0567, Z -7.1667, A 0.000, B 0.000, C 0.000 }
gfCNCPoint5[16787] = {X 110.1220, Y 48.7521, Z -7.1667, A 0.000, B 0.000, C 0.000 }
gfCNCPoint5[16788] = {X 109.3358, Y 48.2612, Z -7.1667, A 0.000, B 0.000, C 0.000 }
gfCNCPoint5[16789] = {X 108.6778, Y 47.6084, Z -7.1667, A 0.000, B 0.000, C 0.000 }
gfCNCPoint5[16790] = {X 108.1807, Y 46.8261, Z -7.1667, A 0.000, B 0.000, C 0.000 }
gfCNCPoint5[16791] = {X 107.8691, Y 45.9531, Z -7.1667, A 0.000, B 0.000, C 0.000 }
gfCNCPoint5[16792] = {X 107.7586, Y 45.0328, Z -7.1667, A 0.000, B 0.000, C 0.000 }
gfCNCPoint5[16793] = {X 107.7585, Y 44.1771, Z -7.1667, A 0.000, B 0.000, C 0.000 }
gfCNCPoint5[16794] = {X 107.7924, Y 43.6576, Z -7.1667, A 0.000, B 0.000, C 0.000 }
gfCNCPoint5[16795] = {X 107.8937, Y 43.1470, Z -7.1667, A 0.000, B 0.000, C 0.000 }
gfCNCPoint5[16796] = {X 108.0559, Y 42.6652, Z -7.1667, A 0.000, B 0.000, C 0.000 }
gfCNCPoint5[16797] = {X 108.2779, Y 42.2079, Z -7.1667, A 0.000, B 0.000, C 0.000 }
gfCNCPoint5[16798] = {X 108.7353, Y 41.5329, Z -7.1667, A 0.000, B 0.000, C 0.000 }
gfCNCPoint5[16799] = {X 109.2849, Y 40.9305, Z -7.1667, A 0.000, B 0.000, C 0.000 }
gfCNCPoint5[16800] = {X 109.2848, Y 39.0829, Z -7.1667, A 0.000, B 0.000, C 0.000 }
gfCNCPoint5[16801] = {X 109.0402, Y 39.0829, Z -7.1667, A 0.000, B 0.000, C 0.000 }
gfCNCPoint5[16802] = {X 105.9641, Y 46.5999, Z -7.1667, A 0.000, B 0.000, C 0.000 }
gfCNCPoint5[16803] = {X 105.6077, Y 47.2737, Z -7.1667, A 0.000, B 0.000, C 0.000 }
gfCNCPoint5[16804] = {X 105.1344, Y 47.8711, Z -7.1667, A 0.000, B 0.000, C 0.000 }
gfCNCPoint5[16805] = {X 104.5601, Y 48.3721, Z -7.1667, A 0.000, B 0.000, C 0.000 }
gfCNCPoint5[16806] = {X 103.9040, Y 48.7600, Z -7.1667, A 0.000, B 0.000, C 0.000 }
gfCNCPoint5[16807] = {X 102.9952, Y 49.0678, Z -7.1667, A 0.000, B 0.000, C 0.000 }
gfCNCPoint5[16808] = {X 102.0400, Y 49.1592, Z -7.1667, A 0.000, B 0.000, C 0.000 }
gfCNCPoint5[16809] = {X 101.0894, Y 49.0293, Z -7.1667, A 0.000, B 0.000, C 0.000 }
gfCNCPoint5[16810] = {X 100.1937, Y 48.6850, Z -7.1667, A 0.000, B 0.000, C 0.000 }
gfCNCPoint5[16811] = {X 99.4008, Y 48.1448, Z -7.1667, A 0.000, B 0.000, C 0.000 }
gfCNCPoint5[16812] = {X 98.7527, Y 47.4372, Z -7.1667, A 0.000, B 0.000, C 0.000 }
gfCNCPoint5[16813] = {X 98.2840, Y 46.5999, Z -7.1667, A 0.000, B 0.000, C 0.000 }
gfCNCPoint5[16814] = {X 94.9720, Y 38.5000, Z -7.1667, A 0.000, B 0.000, C 0.000 }
gfCNCPoint5[16815] = {X 94.9720, Y 40.9788, Z -7.1667, A 0.000, B 0.000, C 0.000 }
gfCNCPoint5[16816] = {X 95.5103, Y 41.5156, Z -7.1667, A 0.000, B 0.000, C 0.000 }
gfCNCPoint5[16817] = {X 95.9439, Y 42.1400, Z -7.1667, A 0.000, B 0.000, C 0.000 }
gfCNCPoint5[16818] = {X 96.1833, Y 42.6321, Z -7.1667, A 0.000, B 0.000, C 0.000 }
gfCNCPoint5[16819] = {X 96.3572, Y 43.1509, Z -7.1667, A 0.000, B 0.000, C 0.000 }
gfCNCPoint5[16820] = {X 96.4613, Y 43.6749, Z -7.1667, A 0.000, B 0.000, C 0.000 }
gfCNCPoint5[16821] = {X 96.4985, Y 44.2078, Z -7.1667, A 0.000, B 0.000, C 0.000 }
gfCNCPoint5[16822] = {X 96.4983, Y 45.0400, Z -7.1667, A 0.000, B 0.000, C 0.000 }
gfCNCPoint5[16823] = {X 96.3865, Y 45.9591, Z -7.1667, A 0.000, B 0.000, C 0.000 }
gfCNCPoint5[16824] = {X 96.0741, Y 46.8306, Z -7.1667, A 0.000, B 0.000, C 0.000 }
gfCNCPoint5[16825] = {X 95.5767, Y 47.6115, Z -7.1667, A 0.000, B 0.000, C 0.000 }
gfCNCPoint5[16826] = {X 94.9188, Y 48.2631, Z -7.1667, A 0.000, B 0.000, C 0.000 }
gfCNCPoint5[16827] = {X 94.1332, Y 48.7530, Z -7.1667, A 0.000, B 0.000, C 0.000 }
gfCNCPoint5[16828] = {X 93.2587, Y 49.0570, Z -7.1667, A 0.000, B 0.000, C 0.000 }
gfCNCPoint5[16829] = {X 92.3385, Y 49.1600, Z -7.1667, A 0.000, B 0.000, C 0.000 }
gfCNCPoint5[16830] = {X 85.8951, Y 49.1600, Z -7.1667, A 0.000, B 0.000, C 0.000 }
gfCNCPoint5[16831] = {X 84.9741, Y 49.0568, Z -7.1667, A 0.000, B 0.000, C 0.000 }
gfCNCPoint5[16832] = {X 84.0988, Y 48.7522, Z -7.1667, A 0.000, B 0.000, C 0.000 }
gfCNCPoint5[16833] = {X 83.3127, Y 48.2614, Z -7.1667, A 0.000, B 0.000, C 0.000 }
gfCNCPoint5[16834] = {X 82.6547, Y 47.6088, Z -7.1667, A 0.000, B 0.000, C 0.000 }
gfCNCPoint5[16835] = {X 82.1576, Y 46.8267, Z -7.1667, A 0.000, B 0.000, C 0.000 }
gfCNCPoint5[16836] = {X 81.8459, Y 45.9539, Z -7.1667, A 0.000, B 0.000, C 0.000 }
gfCNCPoint5[16837] = {X 81.7352, Y 45.0338, Z -7.1667, A 0.000, B 0.000, C 0.000 }
gfCNCPoint5[16838] = {X 81.7351, Y 44.2080, Z -7.1667, A 0.000, B 0.000, C 0.000 }
gfCNCPoint5[16839] = {X 81.8399, Y 43.2948, Z -7.1667, A 0.000, B 0.000, C 0.000 }
gfCNCPoint5[16840] = {X 82.1403, Y 42.4260, Z -7.1667, A 0.000, B 0.000, C 0.000 }
gfCNCPoint5[16841] = {X 82.6219, Y 41.6430, Z -7.1667, A 0.000, B 0.000, C 0.000 }
gfCNCPoint5[16842] = {X 83.2619, Y 40.9830, Z -7.1667, A 0.000, B 0.000, C 0.000 }
gfCNCPoint5[16843] = {X 83.2618, Y 28.5910, Z -7.1667, A 0.000, B 0.000, C 0.000 }
gfCNCPoint5[16844] = {X 79.2618, Y 28.5910, Z -7.1667, A 0.000, B 0.000, C 0.000 }
gfCNCPoint5[16845] = {X 83.3418, Y 28.5910, Z -7.1667, A 0.000, B 0.000, C 0.000 }
gfCNCPoint5[16846] = {X 83.3417, Y 16.1602, Z -7.1667, A 0.000, B 0.000, C 0.000 }
gfCNCPoint5[16847] = {X 82.7049, Y 15.5215, Z -7.1667, A 0.000, B 0.000, C 0.000 }
